KUKA KRL program: EPS_2_25694_LG02A_A_20260223033037.src

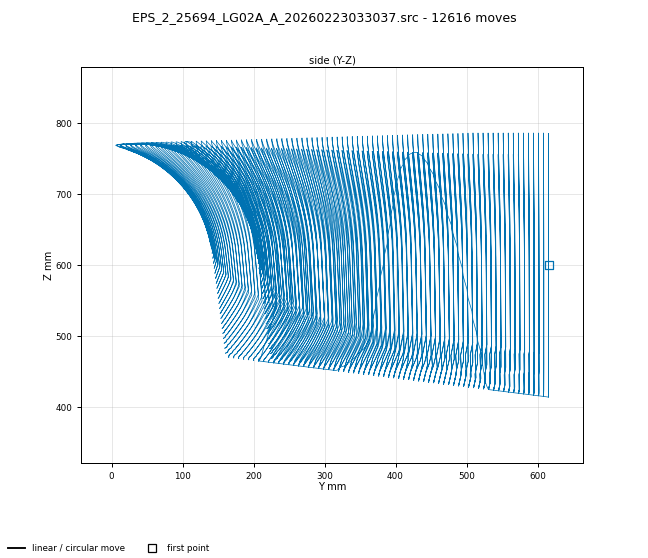
[picture p0: tool path of EPS_2_25694_LG02A_A_20260223033037.src, 12616 of 12618 moves have a stored position in this frame; points joined in program order, loops and branches not executed]
&ACCESS RVP
&REL 4
&COMMENT QRS 19112012
&PARAM EDITMASK = *
DEF PART()
EXT BAS (BAS_COMMAND :IN,REAL :IN )
INT I
BAS (#INITMOV,0 )

;KUKA QRS Post kuka4.cps  Date:22-06-2017 !

File_ID=3041

QRS_PRE_INIT()

;Init var - Until changes are made in qrs_pre_init
Outlet_Square_prg=0
Inlet_1_Square_prg=0
Inlet_2_Square_prg=0
Inlet_3_Square_prg=0
Inlet_4_Square_prg=0
Inlet_5_Square_prg=0

Outlet_1={X 0.000, Y 512.360, Z 637.000, B 0.000, E1 0.000 }
Inlet_1={X 0.000, Y 514.550, Z 607.000, B 0.000, E1 158.000 }
Outlet_1_type=299
Inlet_1_type=299
;QRS#1=Sidecore dimensions
;QRS#2=300-12" PVC SDR 35
;QRS#3=300-12" PVC SDR 35
;QRS#4=
;QRS#5=
;QRS#6=
;QRS#7=
;QRS#8=
;QRS#9=16M PSX
;QRS#10=16M PSX
;QRS#11=
;QRS#12=
;QRS#13=
;QRS#14=
;QRS#15=
;QRS#16=1220x127x1067 3,5'
;QRS#17=EPS Height
;QRS#18=786,5
;QRS#19=*
;QRS#20= UPDATED VERSION 22-06-2017
;QRS#21=*
Outlet_Square=0150
Inlet_1_Square=0150
Inlet_2_Square=0
Inlet_3_Square=0
Inlet_4_Square=0
Inlet_5_Square=0
Mill_Square=1
Outlet_Square_Prg=206
Inlet_1_Square_prg=206

QRS_INIT()

$ADVANCE=5

; T1
PTP {E1 173.596,E2 173.596}
PTP {X 0,Y 615.509,A -85,B 0,C 180,E1 173.596,E2 173.596,E3 0,E4 0,E5 0,E6 0}
QRS_SPEED_INIT()
LIN {X 0,Y 615.509,Z 600,A -85,B 0,C 180,E1 173.596,E2 173.596,E3 0,E4 0,E5 0,E6 0} C_VEL
LIN {X 0,Y 615.509,Z 424.501,A -85,B 0,C 180,E1 173.596,E2 173.596} C_VEL
LIN {X 0,Y 615.509,Z 416.32,A -85,B 0,C 180,E1 173.596,E2 173.596} C_VEL
LIN {X 0,Y 615.491,Z 414.32,A -85,B 0,C 180,E1 173.41,E2 173.41} C_VEL
LIN {X 0,Y 615.479,Z 414.31,A -85,B 0,C 180,E1 170.801,E2 170.801} C_VEL
LIN {X 0,Y 615.485,Z 414.312,A -85,B 0,C 180,E1 168.139,E2 168.139} C_VEL
LIN {X 0,Y 615.494,Z 414.321,A -85,B 0,C 180,E1 165.451,E2 165.451} C_VEL
LIN {X 0,Y 615.478,Z 414.309,A -85,B 0,C 180,E1 162.729,E2 162.729} C_VEL
LIN {X 0,Y 615.483,Z 414.316,A -85,B 0,C 180,E1 159.967,E2 159.967} C_VEL
LIN {X 0,Y 615.482,Z 414.315,A -85,B 0,C 180,E1 157.155,E2 157.155} C_VEL
LIN {X 0,Y 615.495,Z 414.307,A -85,B 0,C 180,E1 154.284,E2 154.284} C_VEL
LIN {X 0,Y 615.491,Z 414.319,A -85,B 0,C 180,E1 151.342,E2 151.342} C_VEL
LIN {X 0,Y 615.477,Z 414.312,A -85,B 0,C 180,E1 148.914,E2 148.914} C_VEL
LIN {X 0,Y 615.485,Z 414.307,A -85,B 0,C 180,E1 146.464,E2 146.464} C_VEL
LIN {X 0,Y 615.491,Z 414.326,A -85,B 0,C 180,E1 143.575,E2 143.575} C_VEL
LIN {X 0,Y 615.479,Z 414.312,A -85,B 0,C 180,E1 140.938,E2 140.938} C_VEL
LIN {X 0,Y 615.482,Z 414.308,A -85,B 0,C 180,E1 138.525,E2 138.525} C_VEL
LIN {X 0,Y 615.484,Z 414.318,A -85,B 0,C 180,E1 135.85,E2 135.85} C_VEL
LIN {X 0,Y 615.492,Z 414.493,A -85,B 0,C 180,E1 134.245,E2 134.245} C_VEL
LIN {X 0,Y 615.492,Z 437.328,A -85,B 0,C 180,E1 131.283,E2 131.283} C_VEL
LIN {X 0,Y 615.491,Z 445.894,A -85,B 0,C 180,E1 130.186,E2 130.186} C_VEL
LIN {X 0,Y 615.498,Z 610.513,A -85,B 0,C 180,E1 128.197,E2 128.197} C_VEL
LIN {X 0,Y 615.48,Z 626.456,A -85,B 0,C 180,E1 127.867,E2 127.867} C_VEL
LIN {X 0,Y 615.485,Z 642.268,A -85,B 0,C 180,E1 127.385,E2 127.385} C_VEL
LIN {X 0,Y 615.486,Z 656.531,A -85,B 0,C 180,E1 126.809,E2 126.809} C_VEL
LIN {X 0,Y 615.498,Z 671.233,A -85,B 0,C 180,E1 126.055,E2 126.055} C_VEL
LIN {X 0,Y 615.497,Z 684.53,A -85,B 0,C 180,E1 125.213,E2 125.213} C_VEL
LIN {X 0,Y 615.497,Z 695.772,A -85,B 0,C 180,E1 124.36,E2 124.36} C_VEL
LIN {X 0,Y 615.497,Z 706.636,A -85,B 0,C 180,E1 123.385,E2 123.385} C_VEL
LIN {X 0,Y 615.496,Z 716.523,A -85,B 0,C 180,E1 122.332,E2 122.332} C_VEL
LIN {X 0,Y 615.497,Z 725.201,A -85,B 0,C 180,E1 121.235,E2 121.235} C_VEL
LIN {X 0,Y 615.497,Z 733.498,A -85,B 0,C 180,E1 119.977,E2 119.977} C_VEL
LIN {X 0,Y 615.493,Z 740.563,A -85,B 0,C 180,E1 118.657,E2 118.657} C_VEL
LIN {X 0,Y 615.496,Z 745.364,A -85,B 0,C 180,E1 117.544,E2 117.544} C_VEL
LIN {X 0,Y 615.49,Z 749.169,A -85,B 0,C 180,E1 116.443,E2 116.443} C_VEL
LIN {X 0,Y 615.491,Z 751.577,A -85,B 0,C 180,E1 115.569,E2 115.569} C_VEL
LIN {X 0,Y 615.495,Z 754.487,A -85,B 0,C 180,E1 114.009,E2 114.009} C_VEL
LIN {X 0,Y 615.491,Z 755.603,A -85,B 0,C 180,E1 112.844,E2 112.844} C_VEL
LIN {X 0,Y 615.494,Z 755.77,A -85,B 0,C 180,E1 111.431,E2 111.431} C_VEL
LIN {X 0,Y 615.492,Z 754.641,A -85,B 0,C 180,E1 110.032,E2 110.032} C_VEL
LIN {X 0,Y 615.488,Z 752.15,A -85,B 0,C 180,E1 108.604,E2 108.604} C_VEL
LIN {X 0,Y 615.49,Z 748.538,A -85,B 0,C 180,E1 107.27,E2 107.27} C_VEL
LIN {X 0,Y 615.495,Z 743.488,A -85,B 0,C 180,E1 105.904,E2 105.904} C_VEL
LIN {X 0,Y 615.492,Z 736.984,A -85,B 0,C 180,E1 104.548,E2 104.548} C_VEL
LIN {X 0,Y 615.494,Z 729.996,A -85,B 0,C 180,E1 103.369,E2 103.369} C_VEL
LIN {X 0,Y 615.494,Z 721.605,A -85,B 0,C 180,E1 102.195,E2 102.195} C_VEL
LIN {X 0,Y 615.499,Z 711.689,A -85,B 0,C 180,E1 101.041,E2 101.041} C_VEL
LIN {X 0,Y 615.497,Z 701.323,A -85,B 0,C 180,E1 100.028,E2 100.028} C_VEL
LIN {X 0,Y 615.497,Z 689.159,A -85,B 0,C 180,E1 99.033,E2 99.033} C_VEL
LIN {X 0,Y 615.498,Z 677.091,A -85,B 0,C 180,E1 98.205,E2 98.205} C_VEL
LIN {X 0,Y 615.482,Z 664.005,A -85,B 0,C 180,E1 97.463,E2 97.463} C_VEL
LIN {X 0,Y 615.493,Z 648.849,A -85,B 0,C 180,E1 96.774,E2 96.774} C_VEL
LIN {X 0,Y 615.487,Z 634.492,A -85,B 0,C 180,E1 96.268,E2 96.268} C_VEL
LIN {X 0,Y 615.499,Z 620.216,A -85,B 0,C 180,E1 95.898,E2 95.898} C_VEL
LIN {X 0,Y 615.479,Z 604.737,A -85,B 0,C 180,E1 95.631,E2 95.631} C_VEL
LIN {X 0,Y 615.479,Z 445.887,A -85,B 0,C 180,E1 93.723,E2 93.723} C_VEL
LIN {X 0,Y 615.493,Z 424.588,A -85,B 0,C 180,E1 90.981,E2 90.981} C_VEL
LIN {X 0,Y 615.478,Z 414.31,A -85,B 0,C 180,E1 89.632,E2 89.632} C_VEL
LIN {X 0,Y 615.476,Z 414.309,A -85,B 0,C 180,E1 87.382,E2 87.382} C_VEL
LIN {X 0,Y 615.488,Z 414.315,A -85,B 0,C 180,E1 84.759,E2 84.759} C_VEL
LIN {X 0,Y 615.496,Z 414.317,A -85,B 0,C 180,E1 82.124,E2 82.124} C_VEL
LIN {X 0,Y 615.476,Z 414.31,A -85,B 0,C 180,E1 79.473,E2 79.473} C_VEL
LIN {X 0,Y 615.493,Z 414.312,A -85,B 0,C 180,E1 76.799,E2 76.799} C_VEL
LIN {X 0,Y 615.495,Z 414.316,A -85,B 0,C 180,E1 74.095,E2 74.095} C_VEL
LIN {X 0,Y 615.477,Z 414.309,A -85,B 0,C 180,E1 71.353,E2 71.353} C_VEL
LIN {X 0,Y 615.494,Z 414.319,A -85,B 0,C 180,E1 68.568,E2 68.568} C_VEL
LIN {X 0,Y 615.488,Z 414.31,A -85,B 0,C 180,E1 65.728,E2 65.728} C_VEL
LIN {X 0,Y 615.491,Z 414.309,A -85,B 0,C 180,E1 62.955,E2 62.955} C_VEL
LIN {X 0,Y 615.494,Z 414.321,A -85,B 0,C 180,E1 60.205,E2 60.205} C_VEL
LIN {X 0,Y 615.481,Z 414.309,A -85,B 0,C 180,E1 57.542,E2 57.542} C_VEL
LIN {X 0,Y 615.478,Z 414.309,A -85,B 0,C 180,E1 55.184,E2 55.184} C_VEL
LIN {X 0,Y 615.494,Z 414.313,A -85,B 0,C 180,E1 52.758,E2 52.758} C_VEL
LIN {X 0,Y 615.494,Z 414.312,A -85,B 0,C 180,E1 49.911,E2 49.911} C_VEL
LIN {X 0,Y 615.49,Z 414.308,A -85,B 0,C 180,E1 47.647,E2 47.647} C_VEL
LIN {X 0,Y 615.482,Z 414.312,A -85,B 0,C 180,E1 44.931,E2 44.931} C_VEL
LIN {X 0,Y 615.49,Z 414.318,A -85,B 0,C 180,E1 42.081,E2 42.081} C_VEL
LIN {X 0,Y 615.498,Z 414.308,A -85,B 0,C 180,E1 39.75,E2 39.75} C_VEL
LIN {X 0,Y 615.479,Z 414.312,A -85,B 0,C 180,E1 36.936,E2 36.936} C_VEL
LIN {X 0,Y 615.493,Z 414.314,A -85,B 0,C 180,E1 34.702,E2 34.702} C_VEL
LIN {X 0,Y 615.488,Z 414.309,A -85,B 0,C 180,E1 31.686,E2 31.686} C_VEL
LIN {X 0,Y 615.482,Z 414.308,A -85,B 0,C 180,E1 29.407,E2 29.407} C_VEL
LIN {X 0,Y 615.478,Z 414.311,A -85,B 0,C 180,E1 27.044,E2 27.044} C_VEL
LIN {X 0,Y 615.492,Z 414.325,A -85,B 0,C 180,E1 24.272,E2 24.272} C_VEL
LIN {X 0,Y 615.486,Z 414.307,A -85,B 0,C 180,E1 21.432,E2 21.432} C_VEL
LIN {X 0,Y 615.494,Z 414.316,A -85,B 0,C 180,E1 18.607,E2 18.607} C_VEL
LIN {X 0,Y 615.487,Z 414.314,A -85,B 0,C 180,E1 15.905,E2 15.905} C_VEL
LIN {X 0,Y 615.478,Z 414.309,A -85,B 0,C 180,E1 13.202,E2 13.202} C_VEL
LIN {X 0,Y 615.494,Z 414.319,A -85,B 0,C 180,E1 10.527,E2 10.527} C_VEL
LIN {X 0,Y 615.486,Z 414.314,A -85,B 0,C 180,E1 7.876,E2 7.876} C_VEL
LIN {X 0,Y 615.481,Z 414.308,A -85,B 0,C 180,E1 5.241,E2 5.241} C_VEL
LIN {X 0,Y 615.491,Z 414.316,A -85,B 0,C 180,E1 2.618,E2 2.618} C_VEL
LIN {X 0,Y 615.486,Z 414.317,A -85,B 0,C 180,E1 0,E2 0} C_VEL
LIN {X 0,Y 615.491,Z 414.306,A -85,B 0,C 180,E1 -2.618,E2 -2.618} C_VEL
LIN {X 0,Y 615.477,Z 414.316,A -85,B 0,C 180,E1 -5.241,E2 -5.241} C_VEL
LIN {X 0,Y 615.489,Z 414.321,A -85,B 0,C 180,E1 -7.875,E2 -7.875} C_VEL
LIN {X 0,Y 615.489,Z 414.307,A -85,B 0,C 180,E1 -10.527,E2 -10.527} C_VEL
LIN {X 0,Y 615.478,Z 414.314,A -85,B 0,C 180,E1 -13.201,E2 -13.201} C_VEL
LIN {X 0,Y 615.487,Z 414.32,A -85,B 0,C 180,E1 -15.905,E2 -15.905} C_VEL
LIN {X 0,Y 615.49,Z 414.306,A -85,B 0,C 180,E1 -18.646,E2 -18.646} C_VEL
LIN {X 0,Y 615.486,Z 414.318,A -85,B 0,C 180,E1 -21.432,E2 -21.432} C_VEL
LIN {X 0,Y 615.481,Z 414.312,A -85,B 0,C 180,E1 -24.272,E2 -24.272} C_VEL
LIN {X 0,Y 615.478,Z 414.311,A -85,B 0,C 180,E1 -27.044,E2 -27.044} C_VEL
LIN {X 0,Y 615.492,Z 414.324,A -85,B 0,C 180,E1 -29.796,E2 -29.796} C_VEL
LIN {X 0,Y 615.485,Z 414.309,A -85,B 0,C 180,E1 -32.458,E2 -32.458} C_VEL
LIN {X 0,Y 615.49,Z 414.306,A -85,B 0,C 180,E1 -34.815,E2 -34.815} C_VEL
LIN {X 0,Y 615.477,Z 414.315,A -85,B 0,C 180,E1 -37.243,E2 -37.243} C_VEL
LIN {X 0,Y 615.478,Z 414.317,A -85,B 0,C 180,E1 -40.088,E2 -40.088} C_VEL
LIN {X 0,Y 615.478,Z 414.312,A -85,B 0,C 180,E1 -42.354,E2 -42.354} C_VEL
LIN {X 0,Y 615.481,Z 414.311,A -85,B 0,C 180,E1 -45.069,E2 -45.069} C_VEL
LIN {X 0,Y 615.488,Z 414.32,A -85,B 0,C 180,E1 -47.92,E2 -47.92} C_VEL
LIN {X 0,Y 615.477,Z 414.314,A -85,B 0,C 180,E1 -50.249,E2 -50.249} C_VEL
LIN {X 0,Y 615.483,Z 414.31,A -85,B 0,C 180,E1 -53.064,E2 -53.064} C_VEL
LIN {X 0,Y 615.487,Z 414.319,A -85,B 0,C 180,E1 -55.978,E2 -55.978} C_VEL
LIN {X 0,Y 615.476,Z 414.313,A -85,B 0,C 180,E1 -58.314,E2 -58.314} C_VEL
LIN {X 0,Y 615.478,Z 414.309,A -85,B 0,C 180,E1 -60.593,E2 -60.593} C_VEL
LIN {X 0,Y 615.492,Z 414.307,A -85,B 0,C 180,E1 -62.954,E2 -62.954} C_VEL
LIN {X 0,Y 615.493,Z 414.437,A -85,B 0,C 180,E1 -64.937,E2 -64.937} C_VEL
LIN {X 0,Y 615.495,Z 440.026,A -85,B 0,C 180,E1 -67.864,E2 -67.864} C_VEL
LIN {X 0,Y 615.49,Z 466.555,A -85,B 0,C 180,E1 -70.835,E2 -70.835} C_VEL
LIN {X 0,Y 615.487,Z 474.978,A -85,B 0,C 180,E1 -71.761,E2 -71.761} C_VEL
LIN {X 0,Y 615.485,Z 641.166,A -85,B 0,C 180,E1 -73.768,E2 -73.768} C_VEL
LIN {X 0,Y 615.487,Z 656.706,A -85,B 0,C 180,E1 -74.095,E2 -74.095} C_VEL
LIN {X 0,Y 615.479,Z 672.046,A -85,B 0,C 180,E1 -74.562,E2 -74.562} C_VEL
LIN {X 0,Y 615.484,Z 685.749,A -85,B 0,C 180,E1 -75.112,E2 -75.112} C_VEL
LIN {X 0,Y 615.493,Z 700.045,A -85,B 0,C 180,E1 -75.833,E2 -75.833} C_VEL
LIN {X 0,Y 615.497,Z 712.896,A -85,B 0,C 180,E1 -76.631,E2 -76.631} C_VEL
LIN {X 0,Y 615.495,Z 725.252,A -85,B 0,C 180,E1 -77.554,E2 -77.554} C_VEL
LIN {X 0,Y 615.495,Z 735.604,A -85,B 0,C 180,E1 -78.473,E2 -78.473} C_VEL
LIN {X 0,Y 615.494,Z 745.182,A -85,B 0,C 180,E1 -79.473,E2 -79.473} C_VEL
LIN {X 0,Y 615.495,Z 754.575,A -85,B 0,C 180,E1 -80.635,E2 -80.635} C_VEL
LIN {X 0,Y 615.495,Z 762.379,A -85,B 0,C 180,E1 -81.794,E2 -81.794} C_VEL
LIN {X 0,Y 615.497,Z 769.606,A -85,B 0,C 180,E1 -83.102,E2 -83.102} C_VEL
LIN {X 0,Y 615.499,Z 775.435,A -85,B 0,C 180,E1 -84.43,E2 -84.43} C_VEL
LIN {X 0,Y 615.491,Z 778.859,A -85,B 0,C 180,E1 -85.415,E2 -85.415} C_VEL
LIN {X 0,Y 615.492,Z 782.317,A -85,B 0,C 180,E1 -86.727,E2 -86.727} C_VEL
LIN {X 0,Y 615.495,Z 784.593,A -85,B 0,C 180,E1 -88.037,E2 -88.037} C_VEL
LIN {X 0,Y 615.493,Z 785.74,A -85,B 0,C 180,E1 -89.345,E2 -89.345} C_VEL
LIN {X 0,Y 615.493,Z 785.741,A -85,B 0,C 180,E1 -90.654,E2 -90.654} C_VEL
LIN {X 0,Y 615.495,Z 784.594,A -85,B 0,C 180,E1 -91.963,E2 -91.963} C_VEL
LIN {X 0,Y 615.492,Z 782.319,A -85,B 0,C 180,E1 -93.273,E2 -93.273} C_VEL
LIN {X 0,Y 615.491,Z 778.862,A -85,B 0,C 180,E1 -94.584,E2 -94.584} C_VEL
LIN {X 0,Y 615.49,Z 774.145,A -85,B 0,C 180,E1 -95.898,E2 -95.898} C_VEL
LIN {X 0,Y 615.496,Z 768.031,A -85,B 0,C 180,E1 -97.215,E2 -97.215} C_VEL
LIN {X 0,Y 615.49,Z 760.336,A -85,B 0,C 180,E1 -98.536,E2 -98.536} C_VEL
LIN {X 0,Y 615.495,Z 752.117,A -85,B 0,C 180,E1 -99.696,E2 -99.696} C_VEL
LIN {X 0,Y 615.496,Z 741.897,A -85,B 0,C 180,E1 -100.892,E2 -100.892} C_VEL
LIN {X 0,Y 615.495,Z 732.073,A -85,B 0,C 180,E1 -101.86,E2 -101.86} C_VEL
LIN {X 0,Y 615.497,Z 719.954,A -85,B 0,C 180,E1 -102.865,E2 -102.865} C_VEL
LIN {X 0,Y 615.498,Z 707.806,A -85,B 0,C 180,E1 -103.705,E2 -103.705} C_VEL
LIN {X 0,Y 615.477,Z 694.388,A -85,B 0,C 180,E1 -104.472,E2 -104.472} C_VEL
LIN {X 0,Y 615.495,Z 679.86,A -85,B 0,C 180,E1 -105.141,E2 -105.141} C_VEL
LIN {X 0,Y 615.477,Z 665.632,A -85,B 0,C 180,E1 -105.65,E2 -105.65} C_VEL
LIN {X 0,Y 615.495,Z 651.159,A -85,B 0,C 180,E1 -106.035,E2 -106.035} C_VEL
LIN {X 0,Y 615.485,Z 636.616,A -85,B 0,C 180,E1 -106.297,E2 -106.297} C_VEL
LIN {X 0,Y 615.49,Z 474.74,A -85,B 0,C 180,E1 -108.259,E2 -108.259} C_VEL
LIN {X 0,Y 615.496,Z 449.397,A -85,B 0,C 180,E1 -111.08,E2 -111.08} C_VEL
LIN {X 0,Y 615.491,Z 423.588,A -85,B 0,C 180,E1 -114.009,E2 -114.009} C_VEL
LIN {X 0,Y 615.491,Z 414.306,A -85,B 0,C 180,E1 -115.099,E2 -115.099} C_VEL
LIN {X 0,Y 615.483,Z 414.317,A -85,B 0,C 180,E1 -117.915,E2 -117.915} C_VEL
LIN {X 0,Y 615.499,Z 414.321,A -85,B 0,C 180,E1 -120.159,E2 -120.159} C_VEL
LIN {X 0,Y 615.487,Z 414.321,A -85,B 0,C 180,E1 -122.457,E2 -122.457} C_VEL
LIN {X 0,Y 615.481,Z 414.313,A -85,B 0,C 180,E1 -124.815,E2 -124.815} C_VEL
LIN {X 0,Y 615.491,Z 414.306,A -85,B 0,C 180,E1 -127.241,E2 -127.241} C_VEL
LIN {X 0,Y 615.489,Z 414.32,A -85,B 0,C 180,E1 -130.089,E2 -130.089} C_VEL
LIN {X 0,Y 615.487,Z 414.308,A -85,B 0,C 180,E1 -133.047,E2 -133.047} C_VEL
LIN {X 0,Y 615.482,Z 414.318,A -85,B 0,C 180,E1 -136.002,E2 -136.002} C_VEL
LIN {X 0,Y 615.479,Z 414.312,A -85,B 0,C 180,E1 -138.905,E2 -138.905} C_VEL
LIN {X 0,Y 615.484,Z 414.308,A -85,B 0,C 180,E1 -141.096,E2 -141.096} C_VEL
LIN {X 0,Y 615.481,Z 414.31,A -85,B 0,C 180,E1 -143.575,E2 -143.575} C_VEL
LIN {X 0,Y 615.479,Z 414.318,A -85,B 0,C 180,E1 -145.978,E2 -145.978} C_VEL
LIN {X 0,Y 615.485,Z 414.328,A -85,B 0,C 180,E1 -148.315,E2 -148.315} C_VEL
LIN {X 0,Y 615.482,Z 414.319,A -85,B 0,C 180,E1 -150.594,E2 -150.594} C_VEL
LIN {X 0,Y 615.478,Z 414.312,A -85,B 0,C 180,E1 -152.955,E2 -152.955} C_VEL
LIN {X 0,Y 615.479,Z 414.312,A -85,B 0,C 180,E1 -155.728,E2 -155.728} C_VEL
LIN {X 0,Y 615.486,Z 414.32,A -85,B 0,C 180,E1 -158.568,E2 -158.568} C_VEL
LIN {X 0,Y 615.492,Z 414.306,A -85,B 0,C 180,E1 -161.391,E2 -161.391} C_VEL
LIN {X 0,Y 615.484,Z 414.319,A -85,B 0,C 180,E1 -164.095,E2 -164.095} C_VEL
LIN {X 0,Y 615.478,Z 414.315,A -85,B 0,C 180,E1 -166.799,E2 -166.799} C_VEL
LIN {X 0,Y 615.489,Z 414.307,A -85,B 0,C 180,E1 -169.473,E2 -169.473} C_VEL
LIN {X 0,Y 615.485,Z 414.32,A -85,B 0,C 180,E1 -172.124,E2 -172.124} C_VEL
LIN {X 0,Y 615.477,Z 414.317,A -85,B 0,C 180,E1 -174.759,E2 -174.759} C_VEL
LIN {X 0,Y 615.491,Z 414.306,A -85,B 0,C 180,E1 -177.382,E2 -177.382} C_VEL
LIN {X 0,Y 615.479,Z 414.317,A -85,B 0,C 180,E1 -180,E2 -180} C_VEL
LIN {X 0,Y 615.491,Z 414.318,A -85,B 0,C 180,E1 -182.618,E2 -182.618} C_VEL
LIN {X 0,Y 615.477,Z 414.31,A -85,B 0,C 180,E1 -185.241,E2 -185.241} C_VEL
LIN {X 0,Y 615.491,Z 414.32,A -85,B 0,C 180,E1 -186.59,E2 -186.59} C_VEL
LIN {X 0,Y 614.807,Z 414.458,A -85,B 0,C 180,E1 -187.136,E2 -187.136} C_VEL
LIN {X 0,Y 611.965,Z 414.879,A -85,B 0,C 180,E1 -188.022,E2 -188.022} C_VEL
LIN {X 0,Y 609.573,Z 415.186,A -85,B 0,C 180,E1 -188.734,E2 -188.734} C_VEL
LIN {X 0,Y 608.541,Z 415.302,A -85,B 0,C 180,E1 -189.284,E2 -189.284} C_VEL
LIN {X 0,Y 608.453,Z 415.312,A -85,B 0,C 180,E1 -189.47,E2 -189.47} C_VEL
LIN {X 0,Y 608.462,Z 415.315,A -85,B 0,C 180,E1 -192,E2 -192} C_VEL
LIN {X 0,Y 608.477,Z 415.314,A -85,B 0,C 180,E1 -194.721,E2 -194.721} C_VEL
LIN {X 0,Y 608.447,Z 415.313,A -85,B 0,C 180,E1 -197.477,E2 -197.477} C_VEL
LIN {X 0,Y 608.464,Z 415.319,A -85,B 0,C 180,E1 -200.274,E2 -200.274} C_VEL
LIN {X 0,Y 608.473,Z 415.32,A -85,B 0,C 180,E1 -202.482,E2 -202.482} C_VEL
LIN {X 0,Y 608.451,Z 415.312,A -85,B 0,C 180,E1 -205.301,E2 -205.301} C_VEL
LIN {X 0,Y 608.445,Z 415.313,A -85,B 0,C 180,E1 -207.518,E2 -207.518} C_VEL
LIN {X 0,Y 608.469,Z 415.313,A -85,B 0,C 180,E1 -209.974,E2 -209.974} C_VEL
LIN {X 0,Y 608.469,Z 415.32,A -85,B 0,C 180,E1 -212.525,E2 -212.525} C_VEL
LIN {X 0,Y 608.449,Z 415.313,A -85,B 0,C 180,E1 -215.278,E2 -215.278} C_VEL
LIN {X 0,Y 608.467,Z 415.318,A -85,B 0,C 180,E1 -218.242,E2 -218.242} C_VEL
LIN {X 0,Y 608.478,Z 415.318,A -85,B 0,C 180,E1 -220.333,E2 -220.333} C_VEL
LIN {X 0,Y 608.464,Z 415.311,A -85,B 0,C 180,E1 -223.309,E2 -223.309} C_VEL
LIN {X 0,Y 608.475,Z 415.41,A -85,B 0,C 180,E1 -225.605,E2 -225.605} C_VEL
LIN {X 0,Y 608.559,Z 433.198,A -85,B 0,C 180,E1 -227.948,E2 -227.948} C_VEL
LIN {X 0,Y 608.526,Z 445.944,A -85,B 0,C 180,E1 -229.602,E2 -229.602} C_VEL
LIN {X 0,Y 608.759,Z 460.794,A -85,B 0,C 180,E1 -229.79,E2 -229.79} C_VEL
LIN {X 0,Y 608.685,Z 611.468,A -85,B 0,C 180,E1 -231.632,E2 -231.632} C_VEL
LIN {X 0,Y 608.638,Z 626.926,A -85,B 0,C 180,E1 -231.962,E2 -231.962} C_VEL
LIN {X 0,Y 608.619,Z 642.036,A -85,B 0,C 180,E1 -232.428,E2 -232.428} C_VEL
LIN {X 0,Y 608.597,Z 656.166,A -85,B 0,C 180,E1 -233.003,E2 -233.003} C_VEL
LIN {X 0,Y 608.573,Z 670.032,A -85,B 0,C 180,E1 -233.712,E2 -233.712} C_VEL
LIN {X 0,Y 608.537,Z 683.04,A -85,B 0,C 180,E1 -234.527,E2 -234.527} C_VEL
LIN {X 0,Y 608.511,Z 694.952,A -85,B 0,C 180,E1 -235.422,E2 -235.422} C_VEL
LIN {X 0,Y 608.503,Z 706.251,A -85,B 0,C 180,E1 -236.432,E2 -236.432} C_VEL
LIN {X 0,Y 608.471,Z 716.109,A -85,B 0,C 180,E1 -237.477,E2 -237.477} C_VEL
LIN {X 0,Y 608.455,Z 726.038,A -85,B 0,C 180,E1 -238.732,E2 -238.732} C_VEL
LIN {X 0,Y 608.463,Z 734.461,A -85,B 0,C 180,E1 -240.03,E2 -240.03} C_VEL
LIN {X 0,Y 608.43,Z 741.587,A -85,B 0,C 180,E1 -241.388,E2 -241.388} C_VEL
LIN {X 0,Y 608.432,Z 747.381,A -85,B 0,C 180,E1 -242.802,E2 -242.802} C_VEL
LIN {X 0,Y 608.429,Z 751.003,A -85,B 0,C 180,E1 -243.964,E2 -243.964} C_VEL
LIN {X 0,Y 608.416,Z 754.237,A -85,B 0,C 180,E1 -245.428,E2 -245.428} C_VEL
LIN {X 0,Y 608.429,Z 756.021,A -85,B 0,C 180,E1 -246.876,E2 -246.876} C_VEL
LIN {X 0,Y 608.415,Z 756.445,A -85,B 0,C 180,E1 -248.307,E2 -248.307} C_VEL
LIN {X 0,Y 608.431,Z 755.551,A -85,B 0,C 180,E1 -249.725,E2 -249.725} C_VEL
LIN {X 0,Y 608.424,Z 753.375,A -85,B 0,C 180,E1 -251.13,E2 -251.13} C_VEL
LIN {X 0,Y 608.425,Z 749.892,A -85,B 0,C 180,E1 -252.523,E2 -252.523} C_VEL
LIN {X 0,Y 608.459,Z 745.057,A -85,B 0,C 180,E1 -253.907,E2 -253.907} C_VEL
LIN {X 0,Y 608.453,Z 738.775,A -85,B 0,C 180,E1 -255.28,E2 -255.28} C_VEL
LIN {X 0,Y 608.46,Z 730.901,A -85,B 0,C 180,E1 -256.644,E2 -256.644} C_VEL
LIN {X 0,Y 608.482,Z 722.538,A -85,B 0,C 180,E1 -257.832,E2 -257.832} C_VEL
LIN {X 0,Y 608.504,Z 712.409,A -85,B 0,C 180,E1 -259.029,E2 -259.029} C_VEL
LIN {X 0,Y 608.492,Z 702.409,A -85,B 0,C 180,E1 -260.024,E2 -260.024} C_VEL
LIN {X 0,Y 608.518,Z 690.408,A -85,B 0,C 180,E1 -261.031,E2 -261.031} C_VEL
LIN {X 0,Y 608.557,Z 677.176,A -85,B 0,C 180,E1 -261.951,E2 -261.951} C_VEL
LIN {X 0,Y 608.585,Z 664.061,A -85,B 0,C 180,E1 -262.703,E2 -262.703} C_VEL
LIN {X 0,Y 608.61,Z 649.663,A -85,B 0,C 180,E1 -263.369,E2 -263.369} C_VEL
LIN {X 0,Y 608.642,Z 634.561,A -85,B 0,C 180,E1 -263.911,E2 -263.911} C_VEL
LIN {X 0,Y 608.695,Z 619.386,A -85,B 0,C 180,E1 -264.306,E2 -264.306} C_VEL
LIN {X 0,Y 608.688,Z 603.326,A -85,B 0,C 180,E1 -264.576,E2 -264.576} C_VEL
LIN {X 0,Y 608.664,Z 446.816,A -85,B 0,C 180,E1 -266.473,E2 -266.473} C_VEL
LIN {X 0,Y 608.518,Z 445.667,A -85,B 0,C 180,E1 -266.524,E2 -266.524} C_VEL
LIN {X 0,Y 608.58,Z 425.315,A -85,B 0,C 180,E1 -269.173,E2 -269.173} C_VEL
LIN {X 0,Y 608.45,Z 415.314,A -85,B 0,C 180,E1 -270.517,E2 -270.517} C_VEL
LIN {X 0,Y 608.485,Z 415.314,A -85,B 0,C 180,E1 -273.311,E2 -273.311} C_VEL
LIN {X 0,Y 608.467,Z 415.315,A -85,B 0,C 180,E1 -275.967,E2 -275.967} C_VEL
LIN {X 0,Y 608.449,Z 415.313,A -85,B 0,C 180,E1 -278.636,E2 -278.636} C_VEL
LIN {X 0,Y 608.484,Z 415.313,A -85,B 0,C 180,E1 -281.324,E2 -281.324} C_VEL
LIN {X 0,Y 608.474,Z 415.314,A -85,B 0,C 180,E1 -284.038,E2 -284.038} C_VEL
LIN {X 0,Y 608.444,Z 415.313,A -85,B 0,C 180,E1 -286.784,E2 -286.784} C_VEL
LIN {X 0,Y 608.46,Z 415.321,A -85,B 0,C 180,E1 -289.57,E2 -289.57} C_VEL
LIN {X 0,Y 608.463,Z 415.311,A -85,B 0,C 180,E1 -292.476,E2 -292.476} C_VEL
LIN {X 0,Y 608.456,Z 415.312,A -85,B 0,C 180,E1 -294.571,E2 -294.571} C_VEL
LIN {X 0,Y 608.483,Z 415.312,A -85,B 0,C 180,E1 -297.208,E2 -297.208} C_VEL
LIN {X 0,Y 608.476,Z 415.314,A -85,B 0,C 180,E1 -299.972,E2 -299.972} C_VEL
LIN {X 0,Y 608.458,Z 415.311,A -85,B 0,C 180,E1 -302.521,E2 -302.521} C_VEL
LIN {X 0,Y 608.445,Z 415.314,A -85,B 0,C 180,E1 -304.904,E2 -304.904} C_VEL
LIN {X 0,Y 608.48,Z 415.311,A -85,B 0,C 180,E1 -307.159,E2 -307.159} C_VEL
LIN {X 0,Y 608.478,Z 415.316,A -85,B 0,C 180,E1 -309.439,E2 -309.439} C_VEL
LIN {X 0,Y 608.462,Z 415.312,A -85,B 0,C 180,E1 -312.334,E2 -312.334} C_VEL
LIN {X 0,Y 608.451,Z 415.312,A -85,B 0,C 180,E1 -314.796,E2 -314.796} C_VEL
LIN {X 0,Y 608.449,Z 415.314,A -85,B 0,C 180,E1 -317.039,E2 -317.039} C_VEL
LIN {X 0,Y 608.458,Z 415.322,A -85,B 0,C 180,E1 -319.697,E2 -319.697} C_VEL
LIN {X 0,Y 608.469,Z 415.312,A -85,B 0,C 180,E1 -322.253,E2 -322.253} C_VEL
LIN {X 0,Y 608.481,Z 415.31,A -85,B 0,C 180,E1 -325.09,E2 -325.09} C_VEL
LIN {X 0,Y 608.473,Z 415.316,A -85,B 0,C 180,E1 -327.906,E2 -327.906} C_VEL
LIN {X 0,Y 608.477,Z 415.311,A -85,B 0,C 180,E1 -330.221,E2 -330.221} C_VEL
LIN {X 0,Y 608.472,Z 415.31,A -85,B 0,C 180,E1 -332.793,E2 -332.793} C_VEL
LIN {X 0,Y 608.453,Z 415.318,A -85,B 0,C 180,E1 -335.429,E2 -335.429} C_VEL
LIN {X 0,Y 608.469,Z 415.311,A -85,B 0,C 180,E1 -338.308,E2 -338.308} C_VEL
LIN {X 0,Y 608.457,Z 415.314,A -85,B 0,C 180,E1 -341.13,E2 -341.13} C_VEL
LIN {X 0,Y 608.465,Z 415.317,A -85,B 0,C 180,E1 -343.906,E2 -343.906} C_VEL
LIN {X 0,Y 608.458,Z 415.311,A -85,B 0,C 180,E1 -346.643,E2 -346.643} C_VEL
LIN {X 0,Y 608.467,Z 415.315,A -85,B 0,C 180,E1 -349.35,E2 -349.35} C_VEL
LIN {X 0,Y 608.479,Z 415.314,A -85,B 0,C 180,E1 -352.033,E2 -352.033} C_VEL
LIN {X 0,Y 608.461,Z 415.311,A -85,B 0,C 180,E1 -354.698,E2 -354.698} C_VEL
LIN {X 0,Y 608.482,Z 415.313,A -85,B 0,C 180,E1 -357.352,E2 -357.352} C_VEL
LIN {X 0,Y 608.476,Z 415.315,A -85,B 0,C 180,E1 -360,E2 -360} C_VEL
LIN {X 0,Y 608.482,Z 415.308,A -85,B 0,C 180,E1 -362.648,E2 -362.648} C_VEL
LIN {X 0,Y 608.458,Z 415.315,A -85,B 0,C 180,E1 -365.302,E2 -365.302} C_VEL
LIN {X 0,Y 608.48,Z 415.315,A -85,B 0,C 180,E1 -367.967,E2 -367.967} C_VEL
LIN {X 0,Y 608.465,Z 415.311,A -85,B 0,C 180,E1 -370.955,E2 -370.955} C_VEL
LIN {X 0,Y 608.459,Z 415.316,A -85,B 0,C 180,E1 -373.356,E2 -373.356} C_VEL
LIN {X 0,Y 608.461,Z 415.315,A -85,B 0,C 180,E1 -376.094,E2 -376.094} C_VEL
LIN {X 0,Y 608.456,Z 415.312,A -85,B 0,C 180,E1 -378.869,E2 -378.869} C_VEL
LIN {X 0,Y 608.466,Z 415.321,A -85,B 0,C 180,E1 -381.691,E2 -381.691} C_VEL
LIN {X 0,Y 608.448,Z 415.313,A -85,B 0,C 180,E1 -384.571,E2 -384.571} C_VEL
LIN {X 0,Y 608.472,Z 415.312,A -85,B 0,C 180,E1 -387.206,E2 -387.206} C_VEL
LIN {X 0,Y 608.468,Z 415.316,A -85,B 0,C 180,E1 -389.972,E2 -389.972} C_VEL
LIN {X 0,Y 608.452,Z 415.312,A -85,B 0,C 180,E1 -392.88,E2 -392.88} C_VEL
LIN {X 0,Y 608.449,Z 415.316,A -85,B 0,C 180,E1 -395.277,E2 -395.277} C_VEL
LIN {X 0,Y 608.464,Z 415.321,A -85,B 0,C 180,E1 -397.747,E2 -397.747} C_VEL
LIN {X 0,Y 608.446,Z 415.315,A -85,B 0,C 180,E1 -400.329,E2 -400.329} C_VEL
LIN {X 0,Y 608.447,Z 415.313,A -85,B 0,C 180,E1 -402.96,E2 -402.96} C_VEL
LIN {X 0,Y 608.46,Z 415.322,A -85,B 0,C 180,E1 -405.736,E2 -405.736} C_VEL
LIN {X 0,Y 608.46,Z 415.311,A -85,B 0,C 180,E1 -408.658,E2 -408.658} C_VEL
LIN {X 0,Y 608.468,Z 415.316,A -85,B 0,C 180,E1 -411.412,E2 -411.412} C_VEL
LIN {X 0,Y 608.445,Z 415.32,A -85,B 0,C 180,E1 -413.955,E2 -413.955} C_VEL
LIN {X 0,Y 608.448,Z 415.315,A -85,B 0,C 180,E1 -416.328,E2 -416.328} C_VEL
LIN {X 0,Y 608.462,Z 415.311,A -85,B 0,C 180,E1 -418.73,E2 -418.73} C_VEL
LIN {X 0,Y 608.47,Z 415.315,A -85,B 0,C 180,E1 -421.381,E2 -421.381} C_VEL
LIN {X 0,Y 608.442,Z 415.322,A -85,B 0,C 180,E1 -423.964,E2 -423.964} C_VEL
LIN {X 0,Y 608.485,Z 415.446,A -85,B 0,C 180,E1 -424.746,E2 -424.746} C_VEL
LIN {X 0,Y 608.662,Z 424.488,A -85,B 0,C 180,E1 -425.809,E2 -425.809} C_VEL
LIN {X 0,Y 608.608,Z 447.83,A -85,B 0,C 180,E1 -428.491,E2 -428.491} C_VEL
LIN {X 0,Y 608.561,Z 471.239,A -85,B 0,C 180,E1 -431.134,E2 -431.134} C_VEL
LIN {X 0,Y 608.577,Z 474.978,A -85,B 0,C 180,E1 -431.547,E2 -431.547} C_VEL
LIN {X 0,Y 608.701,Z 587.844,A -85,B 0,C 180,E1 -432.92,E2 -432.92} C_VEL
LIN {X 0,Y 608.68,Z 641.166,A -85,B 0,C 180,E1 -433.581,E2 -433.581} C_VEL
LIN {X 0,Y 608.647,Z 656.705,A -85,B 0,C 180,E1 -433.911,E2 -433.911} C_VEL
LIN {X 0,Y 608.616,Z 672.044,A -85,B 0,C 180,E1 -434.383,E2 -434.383} C_VEL
LIN {X 0,Y 608.605,Z 685.752,A -85,B 0,C 180,E1 -434.94,E2 -434.94} C_VEL
LIN {X 0,Y 608.572,Z 699.233,A -85,B 0,C 180,E1 -435.624,E2 -435.624} C_VEL
LIN {X 0,Y 608.554,Z 711.661,A -85,B 0,C 180,E1 -436.39,E2 -436.39} C_VEL
LIN {X 0,Y 608.528,Z 724.28,A -85,B 0,C 180,E1 -437.324,E2 -437.324} C_VEL
LIN {X 0,Y 608.496,Z 735.745,A -85,B 0,C 180,E1 -438.339,E2 -438.339} C_VEL
LIN {X 0,Y 608.475,Z 745.386,A -85,B 0,C 180,E1 -439.35,E2 -439.35} C_VEL
LIN {X 0,Y 608.477,Z 754.852,A -85,B 0,C 180,E1 -440.526,E2 -440.526} C_VEL
LIN {X 0,Y 608.456,Z 762.728,A -85,B 0,C 180,E1 -441.698,E2 -441.698} C_VEL
LIN {X 0,Y 608.442,Z 770.086,A -85,B 0,C 180,E1 -443.034,E2 -443.034} C_VEL
LIN {X 0,Y 608.449,Z 775.922,A -85,B 0,C 180,E1 -444.365,E2 -444.365} C_VEL
LIN {X 0,Y 608.427,Z 779.382,A -85,B 0,C 180,E1 -445.362,E2 -445.362} C_VEL
LIN {X 0,Y 608.421,Z 782.885,A -85,B 0,C 180,E1 -446.689,E2 -446.689} C_VEL
LIN {X 0,Y 608.44,Z 785.191,A -85,B 0,C 180,E1 -448.014,E2 -448.014} C_VEL
LIN {X 0,Y 608.436,Z 786.35,A -85,B 0,C 180,E1 -449.338,E2 -449.338} C_VEL
LIN {X 0,Y 608.436,Z 786.351,A -85,B 0,C 180,E1 -450.661,E2 -450.661} C_VEL
LIN {X 0,Y 608.44,Z 785.192,A -85,B 0,C 180,E1 -451.985,E2 -451.985} C_VEL
LIN {X 0,Y 608.421,Z 782.886,A -85,B 0,C 180,E1 -453.311,E2 -453.311} C_VEL
LIN {X 0,Y 608.427,Z 779.384,A -85,B 0,C 180,E1 -454.637,E2 -454.637} C_VEL
LIN {X 0,Y 608.431,Z 774.609,A -85,B 0,C 180,E1 -455.967,E2 -455.967} C_VEL
LIN {X 0,Y 608.458,Z 768.428,A -85,B 0,C 180,E1 -457.299,E2 -457.299} C_VEL
LIN {X 0,Y 608.465,Z 760.657,A -85,B 0,C 180,E1 -458.635,E2 -458.635} C_VEL
LIN {X 0,Y 608.471,Z 752.374,A -85,B 0,C 180,E1 -459.809,E2 -459.809} C_VEL
LIN {X 0,Y 608.492,Z 741.654,A -85,B 0,C 180,E1 -461.063,E2 -461.063} C_VEL
LIN {X 0,Y 608.522,Z 730.28,A -85,B 0,C 180,E1 -462.167,E2 -462.167} C_VEL
LIN {X 0,Y 608.547,Z 718.861,A -85,B 0,C 180,E1 -463.099,E2 -463.099} C_VEL
LIN {X 0,Y 608.561,Z 706.455,A -85,B 0,C 180,E1 -463.95,E2 -463.95} C_VEL
LIN {X 0,Y 608.56,Z 692.87,A -85,B 0,C 180,E1 -464.718,E2 -464.718} C_VEL
LIN {X 0,Y 608.63,Z 678.805,A -85,B 0,C 180,E1 -465.358,E2 -465.358} C_VEL
LIN {X 0,Y 608.631,Z 664.319,A -85,B 0,C 180,E1 -465.874,E2 -465.874} C_VEL
LIN {X 0,Y 608.686,Z 649.039,A -85,B 0,C 180,E1 -466.269,E2 -466.269} C_VEL
LIN {X 0,Y 608.685,Z 633.11,A -85,B 0,C 180,E1 -466.534,E2 -466.534} C_VEL
LIN {X 0,Y 608.686,Z 475.642,A -85,B 0,C 180,E1 -468.442,E2 -468.442} C_VEL
LIN {X 0,Y 608.545,Z 474.565,A -85,B 0,C 180,E1 -468.495,E2 -468.495} C_VEL
LIN {X 0,Y 608.615,Z 449.397,A -85,B 0,C 180,E1 -471.33,E2 -471.33} C_VEL
LIN {X 0,Y 608.684,Z 424.44,A -85,B 0,C 180,E1 -474.196,E2 -474.196} C_VEL
LIN {X 0,Y 608.484,Z 415.453,A -85,B 0,C 180,E1 -475.253,E2 -475.253} C_VEL
LIN {X 0,Y 608.449,Z 415.314,A -85,B 0,C 180,E1 -477.517,E2 -477.517} C_VEL
LIN {X 0,Y 608.466,Z 415.316,A -85,B 0,C 180,E1 -479.971,E2 -479.971} C_VEL
LIN {X 0,Y 608.462,Z 415.318,A -85,B 0,C 180,E1 -482.522,E2 -482.522} C_VEL
LIN {X 0,Y 608.435,Z 415.314,A -85,B 0,C 180,E1 -485.277,E2 -485.277} C_VEL
LIN {X 0,Y 608.47,Z 415.312,A -85,B 0,C 180,E1 -487.745,E2 -487.745} C_VEL
LIN {X 0,Y 608.452,Z 415.323,A -85,B 0,C 180,E1 -490.329,E2 -490.329} C_VEL
LIN {X 0,Y 608.484,Z 415.308,A -85,B 0,C 180,E1 -493.31,E2 -493.31} C_VEL
LIN {X 0,Y 608.466,Z 415.318,A -85,B 0,C 180,E1 -496.13,E2 -496.13} C_VEL
LIN {X 0,Y 608.449,Z 415.315,A -85,B 0,C 180,E1 -498.823,E2 -498.823} C_VEL
LIN {X 0,Y 608.465,Z 415.311,A -85,B 0,C 180,E1 -501.412,E2 -501.412} C_VEL
LIN {X 0,Y 608.472,Z 415.314,A -85,B 0,C 180,E1 -503.95,E2 -503.95} C_VEL
LIN {X 0,Y 608.461,Z 415.322,A -85,B 0,C 180,E1 -506.329,E2 -506.329} C_VEL
LIN {X 0,Y 608.47,Z 415.314,A -85,B 0,C 180,E1 -508.727,E2 -508.727} C_VEL
LIN {X 0,Y 608.471,Z 415.31,A -85,B 0,C 180,E1 -511.378,E2 -511.378} C_VEL
LIN {X 0,Y 608.477,Z 415.319,A -85,B 0,C 180,E1 -514.276,E2 -514.276} C_VEL
LIN {X 0,Y 608.447,Z 415.315,A -85,B 0,C 180,E1 -516.876,E2 -516.876} C_VEL
LIN {X 0,Y 608.459,Z 415.313,A -85,B 0,C 180,E1 -519.726,E2 -519.726} C_VEL
LIN {X 0,Y 608.445,Z 415.321,A -85,B 0,C 180,E1 -522.523,E2 -522.523} C_VEL
LIN {X 0,Y 608.473,Z 415.309,A -85,B 0,C 180,E1 -525.28,E2 -525.28} C_VEL
LIN {X 0,Y 608.46,Z 415.316,A -85,B 0,C 180,E1 -528,E2 -528} C_VEL
LIN {X 0,Y 608.463,Z 415.316,A -85,B 0,C 180,E1 -530.694,E2 -530.694} C_VEL
LIN {X 0,Y 608.469,Z 415.31,A -85,B 0,C 180,E1 -533.368,E2 -533.368} C_VEL
LIN {X 0,Y 608.453,Z 415.317,A -85,B 0,C 180,E1 -536.026,E2 -536.026} C_VEL
LIN {X 0,Y 608.468,Z 415.316,A -85,B 0,C 180,E1 -538.676,E2 -538.676} C_VEL
LIN {X 0,Y 608.468,Z 415.31,A -85,B 0,C 180,E1 -541.324,E2 -541.324} C_VEL
LIN {X 0,Y 608.453,Z 415.316,A -85,B 0,C 180,E1 -543.974,E2 -543.974} C_VEL
LIN {X 0,Y 608.469,Z 415.316,A -85,B 0,C 180,E1 -546.633,E2 -546.633} C_VEL
LIN {X 0,Y 608.453,Z 415.312,A -85,B 0,C 180,E1 -549.47,E2 -549.47} C_VEL
LIN {X 0,Y 607.776,Z 415.402,A -85,B 0,C 180,E1 -550.023,E2 -550.023} C_VEL
LIN {X 0,Y 604.924,Z 415.757,A -85,B 0,C 180,E1 -550.92,E2 -550.92} C_VEL
LIN {X 0,Y 602.522,Z 416.057,A -85,B 0,C 180,E1 -551.641,E2 -551.641} C_VEL
LIN {X 0,Y 601.492,Z 416.186,A -85,B 0,C 180,E1 -552.198,E2 -552.198} C_VEL
LIN {X 0,Y 601.409,Z 416.193,A -85,B 0,C 180,E1 -552.386,E2 -552.386} C_VEL
LIN {X 0,Y 601.429,Z 416.19,A -85,B 0,C 180,E1 -554.897,E2 -554.897} C_VEL
LIN {X 0,Y 601.429,Z 416.189,A -85,B 0,C 180,E1 -556.986,E2 -556.986} C_VEL
LIN {X 0,Y 601.404,Z 416.192,A -85,B 0,C 180,E1 -559.81,E2 -559.81} C_VEL
LIN {X 0,Y 601.418,Z 416.196,A -85,B 0,C 180,E1 -562.608,E2 -562.608} C_VEL
LIN {X 0,Y 601.401,Z 416.194,A -85,B 0,C 180,E1 -564.879,E2 -564.879} C_VEL
LIN {X 0,Y 601.422,Z 416.19,A -85,B 0,C 180,E1 -567.868,E2 -567.868} C_VEL
LIN {X 0,Y 601.443,Z 416.191,A -85,B 0,C 180,E1 -570.163,E2 -570.163} C_VEL
LIN {X 0,Y 601.425,Z 416.194,A -85,B 0,C 180,E1 -572.718,E2 -572.718} C_VEL
LIN {X 0,Y 601.415,Z 416.19,A -85,B 0,C 180,E1 -575.116,E2 -575.116} C_VEL
LIN {X 0,Y 601.43,Z 416.187,A -85,B 0,C 180,E1 -577.42,E2 -577.42} C_VEL
LIN {X 0,Y 601.412,Z 416.193,A -85,B 0,C 180,E1 -579.995,E2 -579.995} C_VEL
LIN {X 0,Y 601.409,Z 416.197,A -85,B 0,C 180,E1 -582.671,E2 -582.671} C_VEL
LIN {X 0,Y 601.45,Z 416.274,A -85,B 0,C 180,E1 -585.445,E2 -585.445} C_VEL
LIN {X 0,Y 601.692,Z 420.354,A -85,B 0,C 180,E1 -586.001,E2 -586.001} C_VEL
LIN {X 0,Y 601.627,Z 442.433,A -85,B 0,C 180,E1 -588.923,E2 -588.923} C_VEL
LIN {X 0,Y 601.594,Z 446.098,A -85,B 0,C 180,E1 -589.383,E2 -589.383} C_VEL
LIN {X 0,Y 602.04,Z 450.336,A -85,B 0,C 180,E1 -589.45,E2 -589.45} C_VEL
LIN {X 0,Y 601.875,Z 611.182,A -85,B 0,C 180,E1 -591.436,E2 -591.436} C_VEL
LIN {X 0,Y 601.819,Z 626.993,A -85,B 0,C 180,E1 -591.776,E2 -591.776} C_VEL
LIN {X 0,Y 601.769,Z 641.813,A -85,B 0,C 180,E1 -592.237,E2 -592.237} C_VEL
LIN {X 0,Y 601.712,Z 656.988,A -85,B 0,C 180,E1 -592.865,E2 -592.865} C_VEL
LIN {X 0,Y 601.658,Z 671.217,A -85,B 0,C 180,E1 -593.612,E2 -593.612} C_VEL
LIN {X 0,Y 601.586,Z 683.971,A -85,B 0,C 180,E1 -594.431,E2 -594.431} C_VEL
LIN {X 0,Y 601.518,Z 696.282,A -85,B 0,C 180,E1 -595.381,E2 -595.381} C_VEL
LIN {X 0,Y 601.487,Z 707.241,A -85,B 0,C 180,E1 -596.39,E2 -596.39} C_VEL
LIN {X 0,Y 601.44,Z 717.279,A -85,B 0,C 180,E1 -597.486,E2 -597.486} C_VEL
LIN {X 0,Y 601.397,Z 725.513,A -85,B 0,C 180,E1 -598.549,E2 -598.549} C_VEL
LIN {X 0,Y 601.385,Z 734.01,A -85,B 0,C 180,E1 -599.859,E2 -599.859} C_VEL
LIN {X 0,Y 601.347,Z 741.195,A -85,B 0,C 180,E1 -601.227,E2 -601.227} C_VEL
LIN {X 0,Y 601.351,Z 745.123,A -85,B 0,C 180,E1 -602.13,E2 -602.13} C_VEL
LIN {X 0,Y 601.349,Z 750.257,A -85,B 0,C 180,E1 -603.634,E2 -603.634} C_VEL
LIN {X 0,Y 601.328,Z 753.776,A -85,B 0,C 180,E1 -605.119,E2 -605.119} C_VEL
LIN {X 0,Y 601.323,Z 755.824,A -85,B 0,C 180,E1 -606.586,E2 -606.586} C_VEL
LIN {X 0,Y 601.336,Z 756.5,A -85,B 0,C 180,E1 -608.039,E2 -608.039} C_VEL
LIN {X 0,Y 601.347,Z 755.847,A -85,B 0,C 180,E1 -609.476,E2 -609.476} C_VEL
LIN {X 0,Y 601.311,Z 753.9,A -85,B 0,C 180,E1 -610.898,E2 -610.898} C_VEL
LIN {X 0,Y 601.316,Z 750.645,A -85,B 0,C 180,E1 -612.31,E2 -612.31} C_VEL
LIN {X 0,Y 601.362,Z 746.051,A -85,B 0,C 180,E1 -613.712,E2 -613.712} C_VEL
LIN {X 0,Y 601.373,Z 740.046,A -85,B 0,C 180,E1 -615.102,E2 -615.102} C_VEL
LIN {X 0,Y 601.381,Z 734.167,A -85,B 0,C 180,E1 -616.205,E2 -616.205} C_VEL
LIN {X 0,Y 601.417,Z 725.695,A -85,B 0,C 180,E1 -617.515,E2 -617.515} C_VEL
LIN {X 0,Y 601.448,Z 716.422,A -85,B 0,C 180,E1 -618.702,E2 -618.702} C_VEL
LIN {X 0,Y 601.483,Z 706.867,A -85,B 0,C 180,E1 -619.736,E2 -619.736} C_VEL
LIN {X 0,Y 601.543,Z 695.697,A -85,B 0,C 180,E1 -620.756,E2 -620.756} C_VEL
LIN {X 0,Y 601.6,Z 683.545,A -85,B 0,C 180,E1 -621.688,E2 -621.688} C_VEL
LIN {X 0,Y 601.654,Z 670.258,A -85,B 0,C 180,E1 -622.534,E2 -622.534} C_VEL
LIN {X 0,Y 601.716,Z 656.795,A -85,B 0,C 180,E1 -623.234,E2 -623.234} C_VEL
LIN {X 0,Y 601.755,Z 642.767,A -85,B 0,C 180,E1 -623.817,E2 -623.817} C_VEL
LIN {X 0,Y 601.833,Z 627.322,A -85,B 0,C 180,E1 -624.304,E2 -624.304} C_VEL
LIN {X 0,Y 601.876,Z 611.93,A -85,B 0,C 180,E1 -624.64,E2 -624.64} C_VEL
LIN {X 0,Y 601.912,Z 558.752,A -85,B 0,C 180,E1 -625.312,E2 -625.312} C_VEL
LIN {X 0,Y 601.938,Z 447.796,A -85,B 0,C 180,E1 -626.675,E2 -626.675} C_VEL
LIN {X 0,Y 601.579,Z 445.741,A -85,B 0,C 180,E1 -626.735,E2 -626.735} C_VEL
LIN {X 0,Y 601.671,Z 424.784,A -85,B 0,C 180,E1 -629.498,E2 -629.498} C_VEL
LIN {X 0,Y 601.492,Z 416.701,A -85,B 0,C 180,E1 -630.586,E2 -630.586} C_VEL
LIN {X 0,Y 601.445,Z 416.189,A -85,B 0,C 180,E1 -630.67,E2 -630.67} C_VEL
LIN {X 0,Y 601.436,Z 416.193,A -85,B 0,C 180,E1 -633.35,E2 -633.35} C_VEL
LIN {X 0,Y 601.418,Z 416.193,A -85,B 0,C 180,E1 -636.037,E2 -636.037} C_VEL
LIN {X 0,Y 601.412,Z 416.19,A -85,B 0,C 180,E1 -638.738,E2 -638.738} C_VEL
LIN {X 0,Y 601.442,Z 416.193,A -85,B 0,C 180,E1 -641.458,E2 -641.458} C_VEL
LIN {X 0,Y 601.424,Z 416.19,A -85,B 0,C 180,E1 -644.206,E2 -644.206} C_VEL
LIN {X 0,Y 601.418,Z 416.19,A -85,B 0,C 180,E1 -646.986,E2 -646.986} C_VEL
LIN {X 0,Y 601.412,Z 416.197,A -85,B 0,C 180,E1 -649.809,E2 -649.809} C_VEL
LIN {X 0,Y 601.416,Z 416.189,A -85,B 0,C 180,E1 -652.683,E2 -652.683} C_VEL
LIN {X 0,Y 601.406,Z 416.19,A -85,B 0,C 180,E1 -654.879,E2 -654.879} C_VEL
LIN {X 0,Y 601.423,Z 416.194,A -85,B 0,C 180,E1 -657.867,E2 -657.867} C_VEL
LIN {X 0,Y 601.433,Z 416.189,A -85,B 0,C 180,E1 -660.164,E2 -660.164} C_VEL
LIN {X 0,Y 601.421,Z 416.188,A -85,B 0,C 180,E1 -662.715,E2 -662.715} C_VEL
LIN {X 0,Y 601.398,Z 416.193,A -85,B 0,C 180,E1 -665.112,E2 -665.112} C_VEL
LIN {X 0,Y 601.439,Z 416.192,A -85,B 0,C 180,E1 -667.419,E2 -667.419} C_VEL
LIN {X 0,Y 601.413,Z 416.194,A -85,B 0,C 180,E1 -669.995,E2 -669.995} C_VEL
LIN {X 0,Y 601.414,Z 416.189,A -85,B 0,C 180,E1 -672.67,E2 -672.67} C_VEL
LIN {X 0,Y 601.428,Z 416.195,A -85,B 0,C 180,E1 -675.482,E2 -675.482} C_VEL
LIN {X 0,Y 601.424,Z 416.188,A -85,B 0,C 180,E1 -678.407,E2 -678.407} C_VEL
LIN {X 0,Y 601.434,Z 416.187,A -85,B 0,C 180,E1 -680.875,E2 -680.875} C_VEL
LIN {X 0,Y 601.445,Z 416.195,A -85,B 0,C 180,E1 -683.734,E2 -683.734} C_VEL
LIN {X 0,Y 601.427,Z 416.187,A -85,B 0,C 180,E1 -686.686,E2 -686.686} C_VEL
LIN {X 0,Y 601.414,Z 416.19,A -85,B 0,C 180,E1 -689.057,E2 -689.057} C_VEL
LIN {X 0,Y 601.439,Z 416.191,A -85,B 0,C 180,E1 -691.373,E2 -691.373} C_VEL
LIN {X 0,Y 601.421,Z 416.191,A -85,B 0,C 180,E1 -694.131,E2 -694.131} C_VEL
LIN {X 0,Y 601.42,Z 416.187,A -85,B 0,C 180,E1 -696.589,E2 -696.589} C_VEL
LIN {X 0,Y 601.435,Z 416.193,A -85,B 0,C 180,E1 -699.478,E2 -699.478} C_VEL
LIN {X 0,Y 601.396,Z 416.192,A -85,B 0,C 180,E1 -702.311,E2 -702.311} C_VEL
LIN {X 0,Y 601.412,Z 416.19,A -85,B 0,C 180,E1 -704.408,E2 -704.408} C_VEL
LIN {X 0,Y 601.422,Z 416.191,A -85,B 0,C 180,E1 -707.172,E2 -707.172} C_VEL
LIN {X 0,Y 601.435,Z 416.193,A -85,B 0,C 180,E1 -709.905,E2 -709.905} C_VEL
LIN {X 0,Y 601.438,Z 416.186,A -85,B 0,C 180,E1 -712.615,E2 -712.615} C_VEL
LIN {X 0,Y 601.429,Z 416.191,A -85,B 0,C 180,E1 -715.308,E2 -715.308} C_VEL
LIN {X 0,Y 601.426,Z 416.193,A -85,B 0,C 180,E1 -717.991,E2 -717.991} C_VEL
LIN {X 0,Y 601.451,Z 416.184,A -85,B 0,C 180,E1 -720.669,E2 -720.669} C_VEL
LIN {X 0,Y 601.428,Z 416.192,A -85,B 0,C 180,E1 -723.349,E2 -723.349} C_VEL
LIN {X 0,Y 601.415,Z 416.193,A -85,B 0,C 180,E1 -726.037,E2 -726.037} C_VEL
LIN {X 0,Y 601.437,Z 416.186,A -85,B 0,C 180,E1 -728.737,E2 -728.737} C_VEL
LIN {X 0,Y 601.433,Z 416.193,A -85,B 0,C 180,E1 -731.458,E2 -731.458} C_VEL
LIN {X 0,Y 601.419,Z 416.191,A -85,B 0,C 180,E1 -734.205,E2 -734.205} C_VEL
LIN {X 0,Y 601.431,Z 416.188,A -85,B 0,C 180,E1 -736.986,E2 -736.986} C_VEL
LIN {X 0,Y 601.404,Z 416.199,A -85,B 0,C 180,E1 -739.809,E2 -739.809} C_VEL
LIN {X 0,Y 601.414,Z 416.189,A -85,B 0,C 180,E1 -742.606,E2 -742.606} C_VEL
LIN {X 0,Y 601.399,Z 416.191,A -85,B 0,C 180,E1 -744.879,E2 -744.879} C_VEL
LIN {X 0,Y 601.419,Z 416.196,A -85,B 0,C 180,E1 -747.867,E2 -747.867} C_VEL
LIN {X 0,Y 601.427,Z 416.191,A -85,B 0,C 180,E1 -750.164,E2 -750.164} C_VEL
LIN {X 0,Y 601.419,Z 416.188,A -85,B 0,C 180,E1 -752.715,E2 -752.715} C_VEL
LIN {X 0,Y 601.415,Z 416.191,A -85,B 0,C 180,E1 -755.115,E2 -755.115} C_VEL
LIN {X 0,Y 601.432,Z 416.192,A -85,B 0,C 180,E1 -757.419,E2 -757.419} C_VEL
LIN {X 0,Y 601.411,Z 416.195,A -85,B 0,C 180,E1 -759.995,E2 -759.995} C_VEL
LIN {X 0,Y 601.408,Z 416.19,A -85,B 0,C 180,E1 -762.671,E2 -762.671} C_VEL
LIN {X 0,Y 601.426,Z 416.194,A -85,B 0,C 180,E1 -765.482,E2 -765.482} C_VEL
LIN {X 0,Y 601.424,Z 416.189,A -85,B 0,C 180,E1 -768.407,E2 -768.407} C_VEL
LIN {X 0,Y 601.434,Z 416.194,A -85,B 0,C 180,E1 -771.529,E2 -771.529} C_VEL
LIN {X 0,Y 601.385,Z 416.195,A -85,B 0,C 180,E1 -774.245,E2 -774.245} C_VEL
LIN {X 0,Y 601.419,Z 416.189,A -85,B 0,C 180,E1 -776.686,E2 -776.686} C_VEL
LIN {X 0,Y 601.424,Z 416.189,A -85,B 0,C 180,E1 -779.058,E2 -779.058} C_VEL
LIN {X 0,Y 601.43,Z 416.192,A -85,B 0,C 180,E1 -781.373,E2 -781.373} C_VEL
LIN {X 0,Y 601.403,Z 416.201,A -85,B 0,C 180,E1 -783.636,E2 -783.636} C_VEL
LIN {X 0,Y 601.426,Z 416.227,A -85,B 0,C 180,E1 -784.521,E2 -784.521} C_VEL
LIN {X 0,Y 601.878,Z 419.738,A -85,B 0,C 180,E1 -784.958,E2 -784.958} C_VEL
LIN {X 0,Y 601.769,Z 443.189,A -85,B 0,C 180,E1 -787.698,E2 -787.698} C_VEL
LIN {X 0,Y 601.668,Z 468.118,A -85,B 0,C 180,E1 -790.555,E2 -790.555} C_VEL
LIN {X 0,Y 601.633,Z 474.862,A -85,B 0,C 180,E1 -791.319,E2 -791.319} C_VEL
LIN {X 0,Y 602.032,Z 478.967,A -85,B 0,C 180,E1 -791.388,E2 -791.388} C_VEL
LIN {X 0,Y 601.875,Z 641.56,A -85,B 0,C 180,E1 -793.398,E2 -793.398} C_VEL
LIN {X 0,Y 601.813,Z 657.481,A -85,B 0,C 180,E1 -793.745,E2 -793.745} C_VEL
LIN {X 0,Y 601.765,Z 672.043,A -85,B 0,C 180,E1 -794.201,E2 -794.201} C_VEL
LIN {X 0,Y 601.719,Z 685.754,A -85,B 0,C 180,E1 -794.764,E2 -794.764} C_VEL
LIN {X 0,Y 601.658,Z 699.229,A -85,B 0,C 180,E1 -795.455,E2 -795.455} C_VEL
LIN {X 0,Y 601.617,Z 712.447,A -85,B 0,C 180,E1 -796.283,E2 -796.283} C_VEL
LIN {X 0,Y 601.531,Z 724.281,A -85,B 0,C 180,E1 -797.174,E2 -797.174} C_VEL
LIN {X 0,Y 601.488,Z 735.745,A -85,B 0,C 180,E1 -798.201,E2 -798.201} C_VEL
LIN {X 0,Y 601.43,Z 745.386,A -85,B 0,C 180,E1 -799.224,E2 -799.224} C_VEL
LIN {X 0,Y 601.428,Z 754.852,A -85,B 0,C 180,E1 -800.414,E2 -800.414} C_VEL
LIN {X 0,Y 601.368,Z 762.728,A -85,B 0,C 180,E1 -801.6,E2 -801.6} C_VEL
LIN {X 0,Y 601.369,Z 770.086,A -85,B 0,C 180,E1 -802.951,E2 -802.951} C_VEL
LIN {X 0,Y 601.371,Z 775.923,A -85,B 0,C 180,E1 -804.299,E2 -804.299} C_VEL
LIN {X 0,Y 601.33,Z 779.382,A -85,B 0,C 180,E1 -805.307,E2 -805.307} C_VEL
LIN {X 0,Y 601.337,Z 782.885,A -85,B 0,C 180,E1 -806.65,E2 -806.65} C_VEL
LIN {X 0,Y 601.339,Z 785.191,A -85,B 0,C 180,E1 -807.99,E2 -807.99} C_VEL
LIN {X 0,Y 601.337,Z 786.35,A -85,B 0,C 180,E1 -809.33,E2 -809.33} C_VEL
LIN {X 0,Y 601.336,Z 786.35,A -85,B 0,C 180,E1 -810.669,E2 -810.669} C_VEL
LIN {X 0,Y 601.339,Z 785.192,A -85,B 0,C 180,E1 -812.009,E2 -812.009} C_VEL
LIN {X 0,Y 601.337,Z 782.887,A -85,B 0,C 180,E1 -813.35,E2 -813.35} C_VEL
LIN {X 0,Y 601.33,Z 779.384,A -85,B 0,C 180,E1 -814.692,E2 -814.692} C_VEL
LIN {X 0,Y 601.352,Z 774.61,A -85,B 0,C 180,E1 -816.037,E2 -816.037} C_VEL
LIN {X 0,Y 601.382,Z 768.428,A -85,B 0,C 180,E1 -817.385,E2 -817.385} C_VEL
LIN {X 0,Y 601.387,Z 760.656,A -85,B 0,C 180,E1 -818.738,E2 -818.738} C_VEL
LIN {X 0,Y 601.427,Z 752.374,A -85,B 0,C 180,E1 -819.925,E2 -819.925} C_VEL
LIN {X 0,Y 601.46,Z 741.935,A -85,B 0,C 180,E1 -821.164,E2 -821.164} C_VEL
LIN {X 0,Y 601.513,Z 732.198,A -85,B 0,C 180,E1 -822.14,E2 -822.14} C_VEL
LIN {X 0,Y 601.57,Z 720.022,A -85,B 0,C 180,E1 -823.168,E2 -823.168} C_VEL
LIN {X 0,Y 601.605,Z 708.085,A -85,B 0,C 180,E1 -824.011,E2 -824.011} C_VEL
LIN {X 0,Y 601.65,Z 694.537,A -85,B 0,C 180,E1 -824.804,E2 -824.804} C_VEL
LIN {X 0,Y 601.761,Z 679.856,A -85,B 0,C 180,E1 -825.495,E2 -825.495} C_VEL
LIN {X 0,Y 601.782,Z 665.635,A -85,B 0,C 180,E1 -826.016,E2 -826.016} C_VEL
LIN {X 0,Y 601.856,Z 650.707,A -85,B 0,C 180,E1 -826.42,E2 -826.42} C_VEL
LIN {X 0,Y 601.867,Z 635.741,A -85,B 0,C 180,E1 -826.689,E2 -826.689} C_VEL
LIN {X 0,Y 601.909,Z 476.419,A -85,B 0,C 180,E1 -828.648,E2 -828.648} C_VEL
LIN {X 0,Y 601.654,Z 474.74,A -85,B 0,C 180,E1 -828.695,E2 -828.695} C_VEL
LIN {X 0,Y 601.74,Z 449.397,A -85,B 0,C 180,E1 -831.586,E2 -831.586} C_VEL
LIN {X 0,Y 601.878,Z 425.303,A -85,B 0,C 180,E1 -834.386,E2 -834.386} C_VEL
LIN {X 0,Y 601.85,Z 418.184,A -85,B 0,C 180,E1 -835.227,E2 -835.227} C_VEL
LIN {X 0,Y 601.421,Z 416.194,A -85,B 0,C 180,E1 -835.501,E2 -835.501} C_VEL
LIN {X 0,Y 601.42,Z 416.194,A -85,B 0,C 180,E1 -837.867,E2 -837.867} C_VEL
LIN {X 0,Y 601.426,Z 416.197,A -85,B 0,C 180,E1 -840.163,E2 -840.163} C_VEL
LIN {X 0,Y 601.422,Z 416.192,A -85,B 0,C 180,E1 -842.716,E2 -842.716} C_VEL
LIN {X 0,Y 601.392,Z 416.192,A -85,B 0,C 180,E1 -845.111,E2 -845.111} C_VEL
LIN {X 0,Y 601.433,Z 416.187,A -85,B 0,C 180,E1 -847.418,E2 -847.418} C_VEL
LIN {X 0,Y 601.409,Z 416.195,A -85,B 0,C 180,E1 -849.994,E2 -849.994} C_VEL
LIN {X 0,Y 601.434,Z 416.191,A -85,B 0,C 180,E1 -852.667,E2 -852.667} C_VEL
LIN {X 0,Y 601.42,Z 416.189,A -85,B 0,C 180,E1 -855.482,E2 -855.482} C_VEL
LIN {X 0,Y 601.419,Z 416.198,A -85,B 0,C 180,E1 -858.406,E2 -858.406} C_VEL
LIN {X 0,Y 601.432,Z 416.189,A -85,B 0,C 180,E1 -860.875,E2 -860.875} C_VEL
LIN {X 0,Y 601.437,Z 416.188,A -85,B 0,C 180,E1 -863.733,E2 -863.733} C_VEL
LIN {X 0,Y 601.429,Z 416.193,A -85,B 0,C 180,E1 -866.063,E2 -866.063} C_VEL
LIN {X 0,Y 601.435,Z 416.193,A -85,B 0,C 180,E1 -868.541,E2 -868.541} C_VEL
LIN {X 0,Y 601.431,Z 416.187,A -85,B 0,C 180,E1 -871.373,E2 -871.373} C_VEL
LIN {X 0,Y 601.417,Z 416.196,A -85,B 0,C 180,E1 -874.13,E2 -874.13} C_VEL
LIN {X 0,Y 601.416,Z 416.195,A -85,B 0,C 180,E1 -876.59,E2 -876.59} C_VEL
LIN {X 0,Y 601.429,Z 416.187,A -85,B 0,C 180,E1 -879.478,E2 -879.478} C_VEL
LIN {X 0,Y 601.392,Z 416.202,A -85,B 0,C 180,E1 -882.312,E2 -882.312} C_VEL
LIN {X 0,Y 601.41,Z 416.199,A -85,B 0,C 180,E1 -884.409,E2 -884.409} C_VEL
LIN {X 0,Y 601.419,Z 416.188,A -85,B 0,C 180,E1 -887.172,E2 -887.172} C_VEL
LIN {X 0,Y 601.433,Z 416.19,A -85,B 0,C 180,E1 -889.905,E2 -889.905} C_VEL
LIN {X 0,Y 601.435,Z 416.193,A -85,B 0,C 180,E1 -892.615,E2 -892.615} C_VEL
LIN {X 0,Y 601.429,Z 416.187,A -85,B 0,C 180,E1 -895.308,E2 -895.308} C_VEL
LIN {X 0,Y 601.423,Z 416.192,A -85,B 0,C 180,E1 -897.991,E2 -897.991} C_VEL
LIN {X 0,Y 601.448,Z 416.19,A -85,B 0,C 180,E1 -900.67,E2 -900.67} C_VEL
LIN {X 0,Y 601.427,Z 416.187,A -85,B 0,C 180,E1 -903.35,E2 -903.35} C_VEL
LIN {X 0,Y 601.431,Z 416.191,A -85,B 0,C 180,E1 -906.037,E2 -906.037} C_VEL
LIN {X 0,Y 601.437,Z 416.191,A -85,B 0,C 180,E1 -908.738,E2 -908.738} C_VEL
LIN {X 0,Y 601.429,Z 416.187,A -85,B 0,C 180,E1 -911.458,E2 -911.458} C_VEL
LIN {X 0,Y 601.409,Z 416.193,A -85,B 0,C 180,E1 -912.386,E2 -912.386} C_VEL
LIN {X 0,Y 600.745,Z 416.275,A -85,B 0,C 180,E1 -912.946,E2 -912.946} C_VEL
LIN {X 0,Y 597.894,Z 416.63,A -85,B 0,C 180,E1 -913.854,E2 -913.854} C_VEL
LIN {X 0,Y 595.482,Z 416.936,A -85,B 0,C 180,E1 -914.584,E2 -914.584} C_VEL
LIN {X 0,Y 594.444,Z 417.059,A -85,B 0,C 180,E1 -915.147,E2 -915.147} C_VEL
LIN {X 0,Y 594.359,Z 417.068,A -85,B 0,C 180,E1 -915.338,E2 -915.338} C_VEL
LIN {X 0,Y 594.376,Z 417.068,A -85,B 0,C 180,E1 -917.905,E2 -917.905} C_VEL
LIN {X 0,Y 594.38,Z 417.068,A -85,B 0,C 180,E1 -920.919,E2 -920.919} C_VEL
LIN {X 0,Y 594.389,Z 417.065,A -85,B 0,C 180,E1 -923.704,E2 -923.704} C_VEL
LIN {X 0,Y 594.383,Z 417.071,A -85,B 0,C 180,E1 -926.7,E2 -926.7} C_VEL
LIN {X 0,Y 594.383,Z 417.067,A -85,B 0,C 180,E1 -928.999,E2 -928.999} C_VEL
LIN {X 0,Y 594.39,Z 417.065,A -85,B 0,C 180,E1 -931.646,E2 -931.646} C_VEL
LIN {X 0,Y 594.395,Z 417.072,A -85,B 0,C 180,E1 -934.579,E2 -934.579} C_VEL
LIN {X 0,Y 594.381,Z 417.067,A -85,B 0,C 180,E1 -937.087,E2 -937.087} C_VEL
LIN {X 0,Y 594.376,Z 417.068,A -85,B 0,C 180,E1 -939.776,E2 -939.776} C_VEL
LIN {X 0,Y 594.367,Z 417.077,A -85,B 0,C 180,E1 -942.376,E2 -942.376} C_VEL
LIN {X 0,Y 594.395,Z 417.111,A -85,B 0,C 180,E1 -945.275,E2 -945.275} C_VEL
LIN {X 0,Y 594.79,Z 420.882,A -85,B 0,C 180,E1 -945.803,E2 -945.803} C_VEL
LIN {X 0,Y 594.659,Z 442.72,A -85,B 0,C 180,E1 -948.728,E2 -948.728} C_VEL
LIN {X 0,Y 594.636,Z 445.904,A -85,B 0,C 180,E1 -949.15,E2 -949.15} C_VEL
LIN {X 0,Y 595.31,Z 450.186,A -85,B 0,C 180,E1 -949.23,E2 -949.23} C_VEL
LIN {X 0,Y 595.095,Z 610.993,A -85,B 0,C 180,E1 -951.238,E2 -951.238} C_VEL
LIN {X 0,Y 594.981,Z 626.865,A -85,B 0,C 180,E1 -951.58,E2 -951.58} C_VEL
LIN {X 0,Y 594.949,Z 641.749,A -85,B 0,C 180,E1 -952.049,E2 -952.049} C_VEL
LIN {X 0,Y 594.847,Z 656.329,A -85,B 0,C 180,E1 -952.654,E2 -952.654} C_VEL
LIN {X 0,Y 594.752,Z 670.572,A -85,B 0,C 180,E1 -953.402,E2 -953.402} C_VEL
LIN {X 0,Y 594.62,Z 684.385,A -85,B 0,C 180,E1 -954.298,E2 -954.298} C_VEL
LIN {X 0,Y 594.53,Z 696.223,A -85,B 0,C 180,E1 -955.225,E2 -955.225} C_VEL
LIN {X 0,Y 594.473,Z 707.192,A -85,B 0,C 180,E1 -956.246,E2 -956.246} C_VEL
LIN {X 0,Y 594.394,Z 718.061,A -85,B 0,C 180,E1 -957.454,E2 -957.454} C_VEL
LIN {X 0,Y 594.353,Z 727.037,A -85,B 0,C 180,E1 -958.65,E2 -958.65} C_VEL
LIN {X 0,Y 594.313,Z 735.129,A -85,B 0,C 180,E1 -959.952,E2 -959.952} C_VEL
LIN {X 0,Y 594.259,Z 740.811,A -85,B 0,C 180,E1 -961.065,E2 -961.065} C_VEL
LIN {X 0,Y 594.268,Z 746.725,A -85,B 0,C 180,E1 -962.496,E2 -962.496} C_VEL
LIN {X 0,Y 594.274,Z 749.382,A -85,B 0,C 180,E1 -963.296,E2 -963.296} C_VEL
LIN {X 0,Y 594.219,Z 753.194,A -85,B 0,C 180,E1 -964.801,E2 -964.801} C_VEL
LIN {X 0,Y 594.223,Z 755.512,A -85,B 0,C 180,E1 -966.29,E2 -966.29} C_VEL
LIN {X 0,Y 594.251,Z 756.441,A -85,B 0,C 180,E1 -967.763,E2 -967.763} C_VEL
LIN {X 0,Y 594.25,Z 756.037,A -85,B 0,C 180,E1 -969.219,E2 -969.219} C_VEL
LIN {X 0,Y 594.21,Z 754.342,A -85,B 0,C 180,E1 -970.661,E2 -970.661} C_VEL
LIN {X 0,Y 594.21,Z 751.349,A -85,B 0,C 180,E1 -972.091,E2 -972.091} C_VEL
LIN {X 0,Y 594.252,Z 747.026,A -85,B 0,C 180,E1 -973.511,E2 -973.511} C_VEL
LIN {X 0,Y 594.29,Z 741.307,A -85,B 0,C 180,E1 -974.92,E2 -974.92} C_VEL
LIN {X 0,Y 594.296,Z 734.067,A -85,B 0,C 180,E1 -976.32,E2 -976.32} C_VEL
LIN {X 0,Y 594.353,Z 726.348,A -85,B 0,C 180,E1 -977.538,E2 -977.538} C_VEL
LIN {X 0,Y 594.417,Z 716.978,A -85,B 0,C 180,E1 -978.765,E2 -978.765} C_VEL
LIN {X 0,Y 594.464,Z 707.761,A -85,B 0,C 180,E1 -979.786,E2 -979.786} C_VEL
LIN {X 0,Y 594.545,Z 695.755,A -85,B 0,C 180,E1 -980.904,E2 -980.904} C_VEL
LIN {X 0,Y 594.648,Z 683.603,A -85,B 0,C 180,E1 -981.847,E2 -981.847} C_VEL
LIN {X 0,Y 594.75,Z 670.313,A -85,B 0,C 180,E1 -982.703,E2 -982.703} C_VEL
LIN {X 0,Y 594.843,Z 655.802,A -85,B 0,C 180,E1 -983.46,E2 -983.46} C_VEL
LIN {X 0,Y 594.952,Z 640.975,A -85,B 0,C 180,E1 -984.068,E2 -984.068} C_VEL
LIN {X 0,Y 595.041,Z 625.75,A -85,B 0,C 180,E1 -984.536,E2 -984.536} C_VEL
LIN {X 0,Y 595.08,Z 610.852,A -85,B 0,C 180,E1 -984.855,E2 -984.855} C_VEL
LIN {X 0,Y 595.198,Z 448.841,A -85,B 0,C 180,E1 -986.88,E2 -986.88} C_VEL
LIN {X 0,Y 594.624,Z 445.822,A -85,B 0,C 180,E1 -986.952,E2 -986.952} C_VEL
LIN {X 0,Y 594.767,Z 425.512,A -85,B 0,C 180,E1 -989.662,E2 -989.662} C_VEL
LIN {X 0,Y 594.574,Z 418.065,A -85,B 0,C 180,E1 -990.678,E2 -990.678} C_VEL
LIN {X 0,Y 594.409,Z 417.068,A -85,B 0,C 180,E1 -990.847,E2 -990.847} C_VEL
LIN {X 0,Y 594.388,Z 417.072,A -85,B 0,C 180,E1 -993.39,E2 -993.39} C_VEL
LIN {X 0,Y 594.368,Z 417.07,A -85,B 0,C 180,E1 -996.109,E2 -996.109} C_VEL
LIN {X 0,Y 594.381,Z 417.066,A -85,B 0,C 180,E1 -998.842,E2 -998.842} C_VEL
LIN {X 0,Y 594.4,Z 417.072,A -85,B 0,C 180,E1 -1001.596,E2 -1001.596} C_VEL
LIN {X 0,Y 594.394,Z 417.064,A -85,B 0,C 180,E1 -1004.377,E2 -1004.377} C_VEL
LIN {X 0,Y 594.385,Z 417.068,A -85,B 0,C 180,E1 -1007.194,E2 -1007.194} C_VEL
LIN {X 0,Y 594.379,Z 417.069,A -85,B 0,C 180,E1 -1010.054,E2 -1010.054} C_VEL
LIN {X 0,Y 594.369,Z 417.068,A -85,B 0,C 180,E1 -1012.967,E2 -1012.967} C_VEL
LIN {X 0,Y 594.381,Z 417.068,A -85,B 0,C 180,E1 -1015.193,E2 -1015.193} C_VEL
LIN {X 0,Y 594.39,Z 417.073,A -85,B 0,C 180,E1 -1017.527,E2 -1017.527} C_VEL
LIN {X 0,Y 594.392,Z 417.065,A -85,B 0,C 180,E1 -1020.328,E2 -1020.328} C_VEL
LIN {X 0,Y 594.381,Z 417.065,A -85,B 0,C 180,E1 -1022.95,E2 -1022.95} C_VEL
LIN {X 0,Y 594.359,Z 417.074,A -85,B 0,C 180,E1 -1025.408,E2 -1025.408} C_VEL
LIN {X 0,Y 594.391,Z 417.069,A -85,B 0,C 180,E1 -1027.94,E2 -1027.94} C_VEL
LIN {X 0,Y 594.38,Z 417.065,A -85,B 0,C 180,E1 -1030.822,E2 -1030.822} C_VEL
LIN {X 0,Y 594.385,Z 417.072,A -85,B 0,C 180,E1 -1033.841,E2 -1033.841} C_VEL
LIN {X 0,Y 594.368,Z 417.067,A -85,B 0,C 180,E1 -1036.7,E2 -1036.7} C_VEL
LIN {X 0,Y 594.374,Z 417.072,A -85,B 0,C 180,E1 -1039.433,E2 -1039.433} C_VEL
LIN {X 0,Y 594.39,Z 417.064,A -85,B 0,C 180,E1 -1042.391,E2 -1042.391} C_VEL
LIN {X 0,Y 594.386,Z 417.064,A -85,B 0,C 180,E1 -1044.671,E2 -1044.671} C_VEL
LIN {X 0,Y 594.38,Z 417.067,A -85,B 0,C 180,E1 -1047.088,E2 -1047.088} C_VEL
LIN {X 0,Y 594.387,Z 417.074,A -85,B 0,C 180,E1 -1049.671,E2 -1049.671} C_VEL
LIN {X 0,Y 594.375,Z 417.066,A -85,B 0,C 180,E1 -1052.539,E2 -1052.539} C_VEL
LIN {X 0,Y 594.378,Z 417.065,A -85,B 0,C 180,E1 -1054.807,E2 -1054.807} C_VEL
LIN {X 0,Y 594.365,Z 417.07,A -85,B 0,C 180,E1 -1057.264,E2 -1057.264} C_VEL
LIN {X 0,Y 594.377,Z 417.071,A -85,B 0,C 180,E1 -1059.946,E2 -1059.946} C_VEL
LIN {X 0,Y 594.39,Z 417.063,A -85,B 0,C 180,E1 -1062.806,E2 -1062.806} C_VEL
LIN {X 0,Y 594.389,Z 417.072,A -85,B 0,C 180,E1 -1065.826,E2 -1065.826} C_VEL
LIN {X 0,Y 594.393,Z 417.064,A -85,B 0,C 180,E1 -1068.404,E2 -1068.404} C_VEL
LIN {X 0,Y 594.399,Z 417.064,A -85,B 0,C 180,E1 -1071.158,E2 -1071.158} C_VEL
LIN {X 0,Y 594.37,Z 417.073,A -85,B 0,C 180,E1 -1073.891,E2 -1073.891} C_VEL
LIN {X 0,Y 594.379,Z 417.064,A -85,B 0,C 180,E1 -1076.61,E2 -1076.61} C_VEL
LIN {X 0,Y 594.42,Z 417.064,A -85,B 0,C 180,E1 -1079.322,E2 -1079.322} C_VEL
LIN {X 0,Y 594.396,Z 417.068,A -85,B 0,C 180,E1 -1082.033,E2 -1082.033} C_VEL
LIN {X 0,Y 594.397,Z 417.061,A -85,B 0,C 180,E1 -1084.747,E2 -1084.747} C_VEL
LIN {X 0,Y 594.392,Z 417.07,A -85,B 0,C 180,E1 -1087.473,E2 -1087.473} C_VEL
LIN {X 0,Y 594.395,Z 417.065,A -85,B 0,C 180,E1 -1090.216,E2 -1090.216} C_VEL
LIN {X 0,Y 594.367,Z 417.067,A -85,B 0,C 180,E1 -1092.983,E2 -1092.983} C_VEL
LIN {X 0,Y 594.366,Z 417.076,A -85,B 0,C 180,E1 -1095.781,E2 -1095.781} C_VEL
LIN {X 0,Y 594.387,Z 417.063,A -85,B 0,C 180,E1 -1098.617,E2 -1098.617} C_VEL
LIN {X 0,Y 594.366,Z 417.074,A -85,B 0,C 180,E1 -1101.503,E2 -1101.503} C_VEL
LIN {X 0,Y 594.387,Z 417.065,A -85,B 0,C 180,E1 -1104.446,E2 -1104.446} C_VEL
LIN {X 0,Y 594.382,Z 417.065,A -85,B 0,C 180,E1 -1106.7,E2 -1106.7} C_VEL
LIN {X 0,Y 594.381,Z 417.066,A -85,B 0,C 180,E1 -1108.998,E2 -1108.998} C_VEL
LIN {X 0,Y 594.376,Z 417.075,A -85,B 0,C 180,E1 -1111.643,E2 -1111.643} C_VEL
LIN {X 0,Y 594.395,Z 417.063,A -85,B 0,C 180,E1 -1114.579,E2 -1114.579} C_VEL
LIN {X 0,Y 594.384,Z 417.066,A -85,B 0,C 180,E1 -1117.087,E2 -1117.087} C_VEL
LIN {X 0,Y 594.376,Z 417.076,A -85,B 0,C 180,E1 -1119.775,E2 -1119.775} C_VEL
LIN {X 0,Y 594.365,Z 417.068,A -85,B 0,C 180,E1 -1122.376,E2 -1122.376} C_VEL
LIN {X 0,Y 594.363,Z 417.07,A -85,B 0,C 180,E1 -1125.191,E2 -1125.191} C_VEL
LIN {X 0,Y 594.371,Z 417.076,A -85,B 0,C 180,E1 -1127.625,E2 -1127.625} C_VEL
LIN {X 0,Y 594.373,Z 417.068,A -85,B 0,C 180,E1 -1130.319,E2 -1130.319} C_VEL
LIN {X 0,Y 594.383,Z 417.065,A -85,B 0,C 180,E1 -1132.913,E2 -1132.913} C_VEL
LIN {X 0,Y 594.381,Z 417.074,A -85,B 0,C 180,E1 -1135.861,E2 -1135.861} C_VEL
LIN {X 0,Y 594.381,Z 417.066,A -85,B 0,C 180,E1 -1138.65,E2 -1138.65} C_VEL
LIN {X 0,Y 594.383,Z 417.067,A -85,B 0,C 180,E1 -1141.042,E2 -1141.042} C_VEL
LIN {X 0,Y 594.383,Z 417.075,A -85,B 0,C 180,E1 -1143.978,E2 -1143.978} C_VEL
LIN {X 0,Y 594.394,Z 417.202,A -85,B 0,C 180,E1 -1144.315,E2 -1144.315} C_VEL
LIN {X 0,Y 595.088,Z 421.299,A -85,B 0,C 180,E1 -1144.839,E2 -1144.839} C_VEL
LIN {X 0,Y 594.91,Z 444.939,A -85,B 0,C 180,E1 -1147.632,E2 -1147.632} C_VEL
LIN {X 0,Y 594.759,Z 469.679,A -85,B 0,C 180,E1 -1150.499,E2 -1150.499} C_VEL
LIN {X 0,Y 594.704,Z 474.88,A -85,B 0,C 180,E1 -1151.095,E2 -1151.095} C_VEL
LIN {X 0,Y 595.313,Z 478.419,A -85,B 0,C 180,E1 -1151.163,E2 -1151.163} C_VEL
LIN {X 0,Y 595.083,Z 641.353,A -85,B 0,C 180,E1 -1153.199,E2 -1153.199} C_VEL
LIN {X 0,Y 595.017,Z 656.703,A -85,B 0,C 180,E1 -1153.532,E2 -1153.532} C_VEL
LIN {X 0,Y 594.931,Z 672.042,A -85,B 0,C 180,E1 -1154.014,E2 -1154.014} C_VEL
LIN {X 0,Y 594.857,Z 685.757,A -85,B 0,C 180,E1 -1154.584,E2 -1154.584} C_VEL
LIN {X 0,Y 594.732,Z 699.231,A -85,B 0,C 180,E1 -1155.281,E2 -1155.281} C_VEL
LIN {X 0,Y 594.681,Z 711.789,A -85,B 0,C 180,E1 -1156.075,E2 -1156.075} C_VEL
LIN {X 0,Y 594.56,Z 724.283,A -85,B 0,C 180,E1 -1157.021,E2 -1157.021} C_VEL
LIN {X 0,Y 594.465,Z 735.746,A -85,B 0,C 180,E1 -1158.059,E2 -1158.059} C_VEL
LIN {X 0,Y 594.388,Z 745.387,A -85,B 0,C 180,E1 -1159.095,E2 -1159.095} C_VEL
LIN {X 0,Y 594.366,Z 754.853,A -85,B 0,C 180,E1 -1160.299,E2 -1160.299} C_VEL
LIN {X 0,Y 594.311,Z 762.729,A -85,B 0,C 180,E1 -1161.499,E2 -1161.499} C_VEL
LIN {X 0,Y 594.293,Z 770.087,A -85,B 0,C 180,E1 -1162.867,E2 -1162.867} C_VEL
LIN {X 0,Y 594.296,Z 775.923,A -85,B 0,C 180,E1 -1164.231,E2 -1164.231} C_VEL
LIN {X 0,Y 594.232,Z 779.383,A -85,B 0,C 180,E1 -1165.251,E2 -1165.251} C_VEL
LIN {X 0,Y 594.257,Z 782.886,A -85,B 0,C 180,E1 -1166.61,E2 -1166.61} C_VEL
LIN {X 0,Y 594.238,Z 785.192,A -85,B 0,C 180,E1 -1167.966,E2 -1167.966} C_VEL
LIN {X 0,Y 594.237,Z 786.35,A -85,B 0,C 180,E1 -1169.322,E2 -1169.322} C_VEL
LIN {X 0,Y 594.237,Z 786.35,A -85,B 0,C 180,E1 -1170.677,E2 -1170.677} C_VEL
LIN {X 0,Y 594.238,Z 785.193,A -85,B 0,C 180,E1 -1172.033,E2 -1172.033} C_VEL
LIN {X 0,Y 594.257,Z 782.887,A -85,B 0,C 180,E1 -1173.39,E2 -1173.39} C_VEL
LIN {X 0,Y 594.232,Z 779.385,A -85,B 0,C 180,E1 -1174.748,E2 -1174.748} C_VEL
LIN {X 0,Y 594.275,Z 774.61,A -85,B 0,C 180,E1 -1176.109,E2 -1176.109} C_VEL
LIN {X 0,Y 594.296,Z 768.427,A -85,B 0,C 180,E1 -1177.474,E2 -1177.474} C_VEL
LIN {X 0,Y 594.331,Z 760.655,A -85,B 0,C 180,E1 -1178.842,E2 -1178.842} C_VEL
LIN {X 0,Y 594.387,Z 752.374,A -85,B 0,C 180,E1 -1180.043,E2 -1180.043} C_VEL
LIN {X 0,Y 594.433,Z 742.561,A -85,B 0,C 180,E1 -1181.231,E2 -1181.231} C_VEL
LIN {X 0,Y 594.53,Z 732.197,A -85,B 0,C 180,E1 -1182.285,E2 -1182.285} C_VEL
LIN {X 0,Y 594.581,Z 720.023,A -85,B 0,C 180,E1 -1183.325,E2 -1183.325} C_VEL
LIN {X 0,Y 594.693,Z 708.083,A -85,B 0,C 180,E1 -1184.177,E2 -1184.177} C_VEL
LIN {X 0,Y 594.75,Z 694.535,A -85,B 0,C 180,E1 -1184.98,E2 -1184.98} C_VEL
LIN {X 0,Y 594.902,Z 679.853,A -85,B 0,C 180,E1 -1185.678,E2 -1185.678} C_VEL
LIN {X 0,Y 594.951,Z 665.634,A -85,B 0,C 180,E1 -1186.204,E2 -1186.204} C_VEL
LIN {X 0,Y 595.048,Z 651.139,A -85,B 0,C 180,E1 -1186.602,E2 -1186.602} C_VEL
LIN {X 0,Y 595.067,Z 635.741,A -85,B 0,C 180,E1 -1186.886,E2 -1186.886} C_VEL
LIN {X 0,Y 595.211,Z 477.72,A -85,B 0,C 180,E1 -1188.849,E2 -1188.849} C_VEL
LIN {X 0,Y 594.732,Z 474.801,A -85,B 0,C 180,E1 -1188.913,E2 -1188.913} C_VEL
LIN {X 0,Y 594.88,Z 450.958,A -85,B 0,C 180,E1 -1191.665,E2 -1191.665} C_VEL
LIN {X 0,Y 595.056,Z 427.548,A -85,B 0,C 180,E1 -1194.416,E2 -1194.416} C_VEL
LIN {X 0,Y 594.983,Z 419.745,A -85,B 0,C 180,E1 -1195.352,E2 -1195.352} C_VEL
LIN {X 0,Y 594.384,Z 417.073,A -85,B 0,C 180,E1 -1195.708,E2 -1195.708} C_VEL
LIN {X 0,Y 594.383,Z 417.077,A -85,B 0,C 180,E1 -1198.226,E2 -1198.226} C_VEL
LIN {X 0,Y 594.386,Z 417.071,A -85,B 0,C 180,E1 -1200.558,E2 -1200.558} C_VEL
LIN {X 0,Y 594.376,Z 417.067,A -85,B 0,C 180,E1 -1202.949,E2 -1202.949} C_VEL
LIN {X 0,Y 594.351,Z 417.069,A -85,B 0,C 180,E1 -1205.408,E2 -1205.408} C_VEL
LIN {X 0,Y 594.386,Z 417.069,A -85,B 0,C 180,E1 -1207.94,E2 -1207.94} C_VEL
LIN {X 0,Y 594.377,Z 417.068,A -85,B 0,C 180,E1 -1210.822,E2 -1210.822} C_VEL
LIN {X 0,Y 594.382,Z 417.065,A -85,B 0,C 180,E1 -1213.297,E2 -1213.297} C_VEL
LIN {X 0,Y 594.362,Z 417.076,A -85,B 0,C 180,E1 -1216.16,E2 -1216.16} C_VEL
LIN {X 0,Y 594.376,Z 417.073,A -85,B 0,C 180,E1 -1218.536,E2 -1218.536} C_VEL
LIN {X 0,Y 594.382,Z 417.065,A -85,B 0,C 180,E1 -1221.295,E2 -1221.295} C_VEL
LIN {X 0,Y 594.39,Z 417.066,A -85,B 0,C 180,E1 -1223.758,E2 -1223.758} C_VEL
LIN {X 0,Y 594.375,Z 417.075,A -85,B 0,C 180,E1 -1226.239,E2 -1226.239} C_VEL
LIN {X 0,Y 594.384,Z 417.07,A -85,B 0,C 180,E1 -1228.651,E2 -1228.651} C_VEL
LIN {X 0,Y 594.38,Z 417.066,A -85,B 0,C 180,E1 -1231.041,E2 -1231.041} C_VEL
LIN {X 0,Y 594.389,Z 417.068,A -85,B 0,C 180,E1 -1233.975,E2 -1233.975} C_VEL
LIN {X 0,Y 594.385,Z 417.075,A -85,B 0,C 180,E1 -1236.296,E2 -1236.296} C_VEL
LIN {X 0,Y 594.401,Z 417.062,A -85,B 0,C 180,E1 -1239.224,E2 -1239.224} C_VEL
LIN {X 0,Y 594.374,Z 417.072,A -85,B 0,C 180,E1 -1242.096,E2 -1242.096} C_VEL
LIN {X 0,Y 594.364,Z 417.075,A -85,B 0,C 180,E1 -1244.219,E2 -1244.219} C_VEL
LIN {X 0,Y 594.365,Z 417.068,A -85,B 0,C 180,E1 -1247.017,E2 -1247.017} C_VEL
LIN {X 0,Y 594.392,Z 417.066,A -85,B 0,C 180,E1 -1249.784,E2 -1249.784} C_VEL
LIN {X 0,Y 594.388,Z 417.072,A -85,B 0,C 180,E1 -1252.527,E2 -1252.527} C_VEL
LIN {X 0,Y 594.396,Z 417.063,A -85,B 0,C 180,E1 -1255.253,E2 -1255.253} C_VEL
LIN {X 0,Y 594.393,Z 417.067,A -85,B 0,C 180,E1 -1257.967,E2 -1257.967} C_VEL
LIN {X 0,Y 594.419,Z 417.065,A -85,B 0,C 180,E1 -1260.678,E2 -1260.678} C_VEL
LIN {X 0,Y 594.378,Z 417.065,A -85,B 0,C 180,E1 -1263.39,E2 -1263.39} C_VEL
LIN {X 0,Y 594.384,Z 417.07,A -85,B 0,C 180,E1 -1266.109,E2 -1266.109} C_VEL
LIN {X 0,Y 594.396,Z 417.067,A -85,B 0,C 180,E1 -1268.842,E2 -1268.842} C_VEL
LIN {X 0,Y 594.389,Z 417.064,A -85,B 0,C 180,E1 -1271.596,E2 -1271.596} C_VEL
LIN {X 0,Y 594.384,Z 417.075,A -85,B 0,C 180,E1 -1274.377,E2 -1274.377} C_VEL
LIN {X 0,Y 594.359,Z 417.068,A -85,B 0,C 180,E1 -1275.338,E2 -1275.338} C_VEL
LIN {X 0,Y 593.689,Z 417.155,A -85,B 0,C 180,E1 -1275.904,E2 -1275.904} C_VEL
LIN {X 0,Y 590.835,Z 417.511,A -85,B 0,C 180,E1 -1276.822,E2 -1276.822} C_VEL
LIN {X 0,Y 588.43,Z 417.813,A -85,B 0,C 180,E1 -1277.561,E2 -1277.561} C_VEL
LIN {X 0,Y 587.403,Z 417.94,A -85,B 0,C 180,E1 -1278.131,E2 -1278.131} C_VEL
LIN {X 0,Y 587.322,Z 417.948,A -85,B 0,C 180,E1 -1278.324,E2 -1278.324} C_VEL
LIN {X 0,Y 587.352,Z 417.942,A -85,B 0,C 180,E1 -1281.045,E2 -1281.045} C_VEL
LIN {X 0,Y 587.334,Z 417.947,A -85,B 0,C 180,E1 -1284.007,E2 -1284.007} C_VEL
LIN {X 0,Y 587.36,Z 417.948,A -85,B 0,C 180,E1 -1286.278,E2 -1286.278} C_VEL
LIN {X 0,Y 587.35,Z 417.942,A -85,B 0,C 180,E1 -1289.135,E2 -1289.135} C_VEL
LIN {X 0,Y 587.354,Z 417.943,A -85,B 0,C 180,E1 -1291.839,E2 -1291.839} C_VEL
LIN {X 0,Y 587.354,Z 417.95,A -85,B 0,C 180,E1 -1294.35,E2 -1294.35} C_VEL
LIN {X 0,Y 587.349,Z 417.947,A -85,B 0,C 180,E1 -1296.747,E2 -1296.747} C_VEL
LIN {X 0,Y 587.344,Z 417.943,A -85,B 0,C 180,E1 -1299.36,E2 -1299.36} C_VEL
LIN {X 0,Y 587.331,Z 417.949,A -85,B 0,C 180,E1 -1302.109,E2 -1302.109} C_VEL
LIN {X 0,Y 587.37,Z 418.037,A -85,B 0,C 180,E1 -1305.115,E2 -1305.115} C_VEL
LIN {X 0,Y 587.91,Z 421.514,A -85,B 0,C 180,E1 -1305.615,E2 -1305.615} C_VEL
LIN {X 0,Y 587.725,Z 443.9,A -85,B 0,C 180,E1 -1308.649,E2 -1308.649} C_VEL
LIN {X 0,Y 587.693,Z 445.906,A -85,B 0,C 180,E1 -1308.918,E2 -1308.918} C_VEL
LIN {X 0,Y 588.596,Z 450.61,A -85,B 0,C 180,E1 -1309.013,E2 -1309.013} C_VEL
LIN {X 0,Y 588.302,Z 610.798,A -85,B 0,C 180,E1 -1311.035,E2 -1311.035} C_VEL
LIN {X 0,Y 588.201,Z 626.455,A -85,B 0,C 180,E1 -1311.374,E2 -1311.374} C_VEL
LIN {X 0,Y 588.103,Z 641.269,A -85,B 0,C 180,E1 -1311.841,E2 -1311.841} C_VEL
LIN {X 0,Y 587.976,Z 655.692,A -85,B 0,C 180,E1 -1312.441,E2 -1312.441} C_VEL
LIN {X 0,Y 587.826,Z 669.288,A -85,B 0,C 180,E1 -1313.153,E2 -1313.153} C_VEL
LIN {X 0,Y 587.72,Z 682.861,A -85,B 0,C 180,E1 -1314.025,E2 -1314.025} C_VEL
LIN {X 0,Y 587.559,Z 696.038,A -85,B 0,C 180,E1 -1315.054,E2 -1315.054} C_VEL
LIN {X 0,Y 587.471,Z 707.146,A -85,B 0,C 180,E1 -1316.098,E2 -1316.098} C_VEL
LIN {X 0,Y 587.364,Z 717.393,A -85,B 0,C 180,E1 -1317.243,E2 -1317.243} C_VEL
LIN {X 0,Y 587.311,Z 726.307,A -85,B 0,C 180,E1 -1318.432,E2 -1318.432} C_VEL
LIN {X 0,Y 587.237,Z 734.967,A -85,B 0,C 180,E1 -1319.825,E2 -1319.825} C_VEL
LIN {X 0,Y 587.187,Z 741.594,A -85,B 0,C 180,E1 -1321.148,E2 -1321.148} C_VEL
LIN {X 0,Y 587.178,Z 747.501,A -85,B 0,C 180,E1 -1322.645,E2 -1322.645} C_VEL
LIN {X 0,Y 587.139,Z 751.126,A -85,B 0,C 180,E1 -1323.864,E2 -1323.864} C_VEL
LIN {X 0,Y 587.148,Z 754.077,A -85,B 0,C 180,E1 -1325.233,E2 -1325.233} C_VEL
LIN {X 0,Y 587.113,Z 755.954,A -85,B 0,C 180,E1 -1326.733,E2 -1326.733} C_VEL
LIN {X 0,Y 587.142,Z 756.467,A -85,B 0,C 180,E1 -1328.219,E2 -1328.219} C_VEL
LIN {X 0,Y 587.118,Z 755.665,A -85,B 0,C 180,E1 -1329.688,E2 -1329.688} C_VEL
LIN {X 0,Y 587.156,Z 753.578,A -85,B 0,C 180,E1 -1331.145,E2 -1331.145} C_VEL
LIN {X 0,Y 587.136,Z 750.186,A -85,B 0,C 180,E1 -1332.588,E2 -1332.588} C_VEL
LIN {X 0,Y 587.193,Z 745.428,A -85,B 0,C 180,E1 -1334.022,E2 -1334.022} C_VEL
LIN {X 0,Y 587.224,Z 739.247,A -85,B 0,C 180,E1 -1335.444,E2 -1335.444} C_VEL
LIN {X 0,Y 587.255,Z 731.512,A -85,B 0,C 180,E1 -1336.857,E2 -1336.857} C_VEL
LIN {X 0,Y 587.342,Z 723.249,A -85,B 0,C 180,E1 -1338.089,E2 -1338.089} C_VEL
LIN {X 0,Y 587.405,Z 713.413,A -85,B 0,C 180,E1 -1339.313,E2 -1339.313} C_VEL
LIN {X 0,Y 587.502,Z 703.411,A -85,B 0,C 180,E1 -1340.359,E2 -1340.359} C_VEL
LIN {X 0,Y 587.604,Z 691.607,A -85,B 0,C 180,E1 -1341.402,E2 -1341.402} C_VEL
LIN {X 0,Y 587.746,Z 678.626,A -85,B 0,C 180,E1 -1342.356,E2 -1342.356} C_VEL
LIN {X 0,Y 587.89,Z 665.771,A -85,B 0,C 180,E1 -1343.135,E2 -1343.135} C_VEL
LIN {X 0,Y 587.986,Z 651.798,A -85,B 0,C 180,E1 -1343.825,E2 -1343.825} C_VEL
LIN {X 0,Y 588.121,Z 637.298,A -85,B 0,C 180,E1 -1344.386,E2 -1344.386} C_VEL
LIN {X 0,Y 588.24,Z 622.306,A -85,B 0,C 180,E1 -1344.817,E2 -1344.817} C_VEL
LIN {X 0,Y 588.287,Z 606.661,A -85,B 0,C 180,E1 -1345.118,E2 -1345.118} C_VEL
LIN {X 0,Y 588.486,Z 449.824,A -85,B 0,C 180,E1 -1347.091,E2 -1347.091} C_VEL
LIN {X 0,Y 587.665,Z 445.907,A -85,B 0,C 180,E1 -1347.173,E2 -1347.173} C_VEL
LIN {X 0,Y 587.864,Z 426.241,A -85,B 0,C 180,E1 -1349.829,E2 -1349.829} C_VEL
LIN {X 0,Y 587.752,Z 420.024,A -85,B 0,C 180,E1 -1350.685,E2 -1350.685} C_VEL
LIN {X 0,Y 587.385,Z 417.944,A -85,B 0,C 180,E1 -1351.007,E2 -1351.007} C_VEL
LIN {X 0,Y 587.34,Z 417.951,A -85,B 0,C 180,E1 -1353.43,E2 -1353.43} C_VEL
LIN {X 0,Y 587.32,Z 417.948,A -85,B 0,C 180,E1 -1356.183,E2 -1356.183} C_VEL
LIN {X 0,Y 587.369,Z 417.941,A -85,B 0,C 180,E1 -1358.255,E2 -1358.255} C_VEL
LIN {X 0,Y 587.353,Z 417.943,A -85,B 0,C 180,E1 -1361.134,E2 -1361.134} C_VEL
LIN {X 0,Y 587.37,Z 417.94,A -85,B 0,C 180,E1 -1364.261,E2 -1364.261} C_VEL
LIN {X 0,Y 587.35,Z 417.948,A -85,B 0,C 180,E1 -1367.406,E2 -1367.406} C_VEL
LIN {X 0,Y 587.331,Z 417.945,A -85,B 0,C 180,E1 -1370.305,E2 -1370.305} C_VEL
LIN {X 0,Y 587.327,Z 417.948,A -85,B 0,C 180,E1 -1373.259,E2 -1373.259} C_VEL
LIN {X 0,Y 587.34,Z 417.95,A -85,B 0,C 180,E1 -1375.516,E2 -1375.516} C_VEL
LIN {X 0,Y 587.352,Z 417.948,A -85,B 0,C 180,E1 -1377.818,E2 -1377.818} C_VEL
LIN {X 0,Y 587.346,Z 417.942,A -85,B 0,C 180,E1 -1380.511,E2 -1380.511} C_VEL
LIN {X 0,Y 587.343,Z 417.943,A -85,B 0,C 180,E1 -1383.112,E2 -1383.112} C_VEL
LIN {X 0,Y 587.35,Z 417.947,A -85,B 0,C 180,E1 -1385.896,E2 -1385.896} C_VEL
LIN {X 0,Y 587.336,Z 417.942,A -85,B 0,C 180,E1 -1388.479,E2 -1388.479} C_VEL
LIN {X 0,Y 587.34,Z 417.945,A -85,B 0,C 180,E1 -1391.157,E2 -1391.157} C_VEL
LIN {X 0,Y 587.337,Z 417.946,A -85,B 0,C 180,E1 -1394.114,E2 -1394.114} C_VEL
LIN {X 0,Y 587.317,Z 417.946,A -85,B 0,C 180,E1 -1396.993,E2 -1396.993} C_VEL
LIN {X 0,Y 587.322,Z 417.954,A -85,B 0,C 180,E1 -1399.746,E2 -1399.746} C_VEL
LIN {X 0,Y 587.346,Z 417.942,A -85,B 0,C 180,E1 -1402.392,E2 -1402.392} C_VEL
LIN {X 0,Y 587.351,Z 417.941,A -85,B 0,C 180,E1 -1404.946,E2 -1404.946} C_VEL
LIN {X 0,Y 587.341,Z 417.948,A -85,B 0,C 180,E1 -1407.421,E2 -1407.421} C_VEL
LIN {X 0,Y 587.335,Z 417.95,A -85,B 0,C 180,E1 -1409.83,E2 -1409.83} C_VEL
LIN {X 0,Y 587.353,Z 417.942,A -85,B 0,C 180,E1 -1412.307,E2 -1412.307} C_VEL
LIN {X 0,Y 587.339,Z 417.942,A -85,B 0,C 180,E1 -1414.483,E2 -1414.483} C_VEL
LIN {X 0,Y 587.341,Z 417.948,A -85,B 0,C 180,E1 -1417.486,E2 -1417.486} C_VEL
LIN {X 0,Y 587.344,Z 417.942,A -85,B 0,C 180,E1 -1420.425,E2 -1420.425} C_VEL
LIN {X 0,Y 587.355,Z 417.944,A -85,B 0,C 180,E1 -1423.311,E2 -1423.311} C_VEL
LIN {X 0,Y 587.358,Z 417.943,A -85,B 0,C 180,E1 -1426.154,E2 -1426.154} C_VEL
LIN {X 0,Y 587.342,Z 417.942,A -85,B 0,C 180,E1 -1428.962,E2 -1428.962} C_VEL
LIN {X 0,Y 587.371,Z 417.948,A -85,B 0,C 180,E1 -1431.745,E2 -1431.745} C_VEL
LIN {X 0,Y 587.355,Z 417.94,A -85,B 0,C 180,E1 -1434.507,E2 -1434.507} C_VEL
LIN {X 0,Y 587.377,Z 417.94,A -85,B 0,C 180,E1 -1437.257,E2 -1437.257} C_VEL
LIN {X 0,Y 587.382,Z 417.942,A -85,B 0,C 180,E1 -1440,E2 -1440} C_VEL
LIN {X 0,Y 587.377,Z 417.937,A -85,B 0,C 180,E1 -1442.743,E2 -1442.743} C_VEL
LIN {X 0,Y 587.353,Z 417.945,A -85,B 0,C 180,E1 -1445.493,E2 -1445.493} C_VEL
LIN {X 0,Y 587.371,Z 417.94,A -85,B 0,C 180,E1 -1448.255,E2 -1448.255} C_VEL
LIN {X 0,Y 587.347,Z 417.943,A -85,B 0,C 180,E1 -1451.134,E2 -1451.134} C_VEL
LIN {X 0,Y 587.364,Z 417.941,A -85,B 0,C 180,E1 -1454.26,E2 -1454.26} C_VEL
LIN {X 0,Y 587.349,Z 417.946,A -85,B 0,C 180,E1 -1457.406,E2 -1457.406} C_VEL
LIN {X 0,Y 587.329,Z 417.945,A -85,B 0,C 180,E1 -1460.305,E2 -1460.305} C_VEL
LIN {X 0,Y 587.321,Z 417.948,A -85,B 0,C 180,E1 -1463.259,E2 -1463.259} C_VEL
LIN {X 0,Y 587.337,Z 417.95,A -85,B 0,C 180,E1 -1465.516,E2 -1465.516} C_VEL
LIN {X 0,Y 587.348,Z 417.95,A -85,B 0,C 180,E1 -1467.818,E2 -1467.818} C_VEL
LIN {X 0,Y 587.335,Z 417.943,A -85,B 0,C 180,E1 -1470.51,E2 -1470.51} C_VEL
LIN {X 0,Y 587.334,Z 417.948,A -85,B 0,C 180,E1 -1473.397,E2 -1473.397} C_VEL
LIN {X 0,Y 587.356,Z 417.948,A -85,B 0,C 180,E1 -1475.895,E2 -1475.895} C_VEL
LIN {X 0,Y 587.33,Z 417.944,A -85,B 0,C 180,E1 -1478.479,E2 -1478.479} C_VEL
LIN {X 0,Y 587.334,Z 417.945,A -85,B 0,C 180,E1 -1481.157,E2 -1481.157} C_VEL
LIN {X 0,Y 587.326,Z 417.948,A -85,B 0,C 180,E1 -1484.113,E2 -1484.113} C_VEL
LIN {X 0,Y 587.323,Z 417.945,A -85,B 0,C 180,E1 -1486.994,E2 -1486.994} C_VEL
LIN {X 0,Y 587.314,Z 417.956,A -85,B 0,C 180,E1 -1489.746,E2 -1489.746} C_VEL
LIN {X 0,Y 587.346,Z 417.943,A -85,B 0,C 180,E1 -1492.392,E2 -1492.392} C_VEL
LIN {X 0,Y 587.361,Z 417.95,A -85,B 0,C 180,E1 -1495.78,E2 -1495.78} C_VEL
LIN {X 0,Y 587.348,Z 417.945,A -85,B 0,C 180,E1 -1498.231,E2 -1498.231} C_VEL
LIN {X 0,Y 587.349,Z 417.943,A -85,B 0,C 180,E1 -1500.867,E2 -1500.867} C_VEL
LIN {X 0,Y 587.359,Z 417.95,A -85,B 0,C 180,E1 -1503.819,E2 -1503.819} C_VEL
LIN {X 0,Y 587.389,Z 418.178,A -85,B 0,C 180,E1 -1504.105,E2 -1504.105} C_VEL
LIN {X 0,Y 588.289,Z 423.016,A -85,B 0,C 180,E1 -1504.736,E2 -1504.736} C_VEL
LIN {X 0,Y 588.055,Z 446.269,A -85,B 0,C 180,E1 -1507.515,E2 -1507.515} C_VEL
LIN {X 0,Y 587.843,Z 471.239,A -85,B 0,C 180,E1 -1510.442,E2 -1510.442} C_VEL
LIN {X 0,Y 587.811,Z 475.138,A -85,B 0,C 180,E1 -1510.872,E2 -1510.872} C_VEL
LIN {X 0,Y 588.596,Z 479.512,A -85,B 0,C 180,E1 -1510.954,E2 -1510.954} C_VEL
LIN {X 0,Y 588.303,Z 641.318,A -85,B 0,C 180,E1 -1512.998,E2 -1512.998} C_VEL
LIN {X 0,Y 588.211,Z 656.702,A -85,B 0,C 180,E1 -1513.336,E2 -1513.336} C_VEL
LIN {X 0,Y 588.069,Z 672.04,A -85,B 0,C 180,E1 -1513.823,E2 -1513.823} C_VEL
LIN {X 0,Y 587.987,Z 685.759,A -85,B 0,C 180,E1 -1514.399,E2 -1514.399} C_VEL
LIN {X 0,Y 587.829,Z 699.234,A -85,B 0,C 180,E1 -1515.105,E2 -1515.105} C_VEL
LIN {X 0,Y 587.741,Z 712.11,A -85,B 0,C 180,E1 -1515.929,E2 -1515.929} C_VEL
LIN {X 0,Y 587.582,Z 724.284,A -85,B 0,C 180,E1 -1516.864,E2 -1516.864} C_VEL
LIN {X 0,Y 587.454,Z 735.746,A -85,B 0,C 180,E1 -1517.915,E2 -1517.915} C_VEL
LIN {X 0,Y 587.348,Z 745.388,A -85,B 0,C 180,E1 -1518.962,E2 -1518.962} C_VEL
LIN {X 0,Y 587.305,Z 754.854,A -85,B 0,C 180,E1 -1520.182,E2 -1520.182} C_VEL
LIN {X 0,Y 587.264,Z 762.73,A -85,B 0,C 180,E1 -1521.396,E2 -1521.396} C_VEL
LIN {X 0,Y 587.216,Z 770.087,A -85,B 0,C 180,E1 -1522.78,E2 -1522.78} C_VEL
LIN {X 0,Y 587.224,Z 775.923,A -85,B 0,C 180,E1 -1524.161,E2 -1524.161} C_VEL
LIN {X 0,Y 587.136,Z 779.383,A -85,B 0,C 180,E1 -1525.193,E2 -1525.193} C_VEL
LIN {X 0,Y 587.179,Z 782.887,A -85,B 0,C 180,E1 -1526.569,E2 -1526.569} C_VEL
LIN {X 0,Y 587.137,Z 785.193,A -85,B 0,C 180,E1 -1527.942,E2 -1527.942} C_VEL
LIN {X 0,Y 587.137,Z 786.35,A -85,B 0,C 180,E1 -1529.314,E2 -1529.314} C_VEL
LIN {X 0,Y 587.137,Z 786.35,A -85,B 0,C 180,E1 -1530.685,E2 -1530.685} C_VEL
LIN {X 0,Y 587.137,Z 785.193,A -85,B 0,C 180,E1 -1532.058,E2 -1532.058} C_VEL
LIN {X 0,Y 587.179,Z 782.887,A -85,B 0,C 180,E1 -1533.431,E2 -1533.431} C_VEL
LIN {X 0,Y 587.136,Z 779.385,A -85,B 0,C 180,E1 -1534.806,E2 -1534.806} C_VEL
LIN {X 0,Y 587.178,Z 774.61,A -85,B 0,C 180,E1 -1536.184,E2 -1536.184} C_VEL
LIN {X 0,Y 587.235,Z 768.427,A -85,B 0,C 180,E1 -1537.564,E2 -1537.564} C_VEL
LIN {X 0,Y 587.266,Z 760.654,A -85,B 0,C 180,E1 -1538.95,E2 -1538.95} C_VEL
LIN {X 0,Y 587.351,Z 752.373,A -85,B 0,C 180,E1 -1540.165,E2 -1540.165} C_VEL
LIN {X 0,Y 587.399,Z 742.399,A -85,B 0,C 180,E1 -1541.385,E2 -1541.385} C_VEL
LIN {X 0,Y 587.521,Z 732.196,A -85,B 0,C 180,E1 -1542.434,E2 -1542.434} C_VEL
LIN {X 0,Y 587.629,Z 720.024,A -85,B 0,C 180,E1 -1543.486,E2 -1543.486} C_VEL
LIN {X 0,Y 587.773,Z 707.064,A -85,B 0,C 180,E1 -1544.416,E2 -1544.416} C_VEL
LIN {X 0,Y 587.886,Z 692.876,A -85,B 0,C 180,E1 -1545.248,E2 -1545.248} C_VEL
LIN {X 0,Y 588.049,Z 678.81,A -85,B 0,C 180,E1 -1545.91,E2 -1545.91} C_VEL
LIN {X 0,Y 588.168,Z 664.321,A -85,B 0,C 180,E1 -1546.441,E2 -1546.441} C_VEL
LIN {X 0,Y 588.278,Z 649.297,A -85,B 0,C 180,E1 -1546.844,E2 -1546.844} C_VEL
LIN {X 0,Y 588.32,Z 634.107,A -85,B 0,C 180,E1 -1547.11,E2 -1547.11} C_VEL
LIN {X 0,Y 588.501,Z 478.542,A -85,B 0,C 180,E1 -1549.062,E2 -1549.062} C_VEL
LIN {X 0,Y 587.805,Z 474.774,A -85,B 0,C 180,E1 -1549.148,E2 -1549.148} C_VEL
LIN {X 0,Y 588.008,Z 450.958,A -85,B 0,C 180,E1 -1551.931,E2 -1551.931} C_VEL
LIN {X 0,Y 588.258,Z 427.092,A -85,B 0,C 180,E1 -1554.772,E2 -1554.772} C_VEL
LIN {X 0,Y 588.117,Z 421.306,A -85,B 0,C 180,E1 -1555.48,E2 -1555.48} C_VEL
LIN {X 0,Y 587.338,Z 417.952,A -85,B 0,C 180,E1 -1555.949,E2 -1555.949} C_VEL
LIN {X 0,Y 587.325,Z 417.951,A -85,B 0,C 180,E1 -1558.596,E2 -1558.596} C_VEL
LIN {X 0,Y 587.339,Z 417.944,A -85,B 0,C 180,E1 -1560.965,E2 -1560.965} C_VEL
LIN {X 0,Y 587.332,Z 417.944,A -85,B 0,C 180,E1 -1563.396,E2 -1563.396} C_VEL
LIN {X 0,Y 587.315,Z 417.95,A -85,B 0,C 180,E1 -1565.897,E2 -1565.897} C_VEL
LIN {X 0,Y 587.33,Z 417.951,A -85,B 0,C 180,E1 -1568.478,E2 -1568.478} C_VEL
LIN {X 0,Y 587.333,Z 417.944,A -85,B 0,C 180,E1 -1571.156,E2 -1571.156} C_VEL
LIN {X 0,Y 587.329,Z 417.951,A -85,B 0,C 180,E1 -1574.114,E2 -1574.114} C_VEL
LIN {X 0,Y 587.309,Z 417.947,A -85,B 0,C 180,E1 -1576.993,E2 -1576.993} C_VEL
LIN {X 0,Y 587.314,Z 417.948,A -85,B 0,C 180,E1 -1579.746,E2 -1579.746} C_VEL
LIN {X 0,Y 587.338,Z 417.952,A -85,B 0,C 180,E1 -1582.392,E2 -1582.392} C_VEL
LIN {X 0,Y 587.347,Z 417.943,A -85,B 0,C 180,E1 -1584.946,E2 -1584.946} C_VEL
LIN {X 0,Y 587.334,Z 417.943,A -85,B 0,C 180,E1 -1587.421,E2 -1587.421} C_VEL
LIN {X 0,Y 587.328,Z 417.946,A -85,B 0,C 180,E1 -1589.83,E2 -1589.83} C_VEL
LIN {X 0,Y 587.344,Z 417.952,A -85,B 0,C 180,E1 -1592.306,E2 -1592.306} C_VEL
LIN {X 0,Y 587.335,Z 417.951,A -85,B 0,C 180,E1 -1594.484,E2 -1594.484} C_VEL
LIN {X 0,Y 587.333,Z 417.943,A -85,B 0,C 180,E1 -1597.486,E2 -1597.486} C_VEL
LIN {X 0,Y 587.326,Z 417.945,A -85,B 0,C 180,E1 -1599.695,E2 -1599.695} C_VEL
LIN {X 0,Y 587.351,Z 417.947,A -85,B 0,C 180,E1 -1602.594,E2 -1602.594} C_VEL
LIN {X 0,Y 587.357,Z 417.942,A -85,B 0,C 180,E1 -1605.739,E2 -1605.739} C_VEL
LIN {X 0,Y 587.336,Z 417.951,A -85,B 0,C 180,E1 -1608.263,E2 -1608.263} C_VEL
LIN {X 0,Y 587.34,Z 417.943,A -85,B 0,C 180,E1 -1611.051,E2 -1611.051} C_VEL
LIN {X 0,Y 587.368,Z 417.939,A -85,B 0,C 180,E1 -1613.264,E2 -1613.264} C_VEL
LIN {X 0,Y 587.316,Z 417.948,A -85,B 0,C 180,E1 -1615.883,E2 -1615.883} C_VEL
LIN {X 0,Y 587.363,Z 417.943,A -85,B 0,C 180,E1 -1617.943,E2 -1617.943} C_VEL
LIN {X 0,Y 587.389,Z 417.941,A -85,B 0,C 180,E1 -1620.686,E2 -1620.686} C_VEL
LIN {X 0,Y 587.33,Z 417.944,A -85,B 0,C 180,E1 -1623.43,E2 -1623.43} C_VEL
LIN {X 0,Y 587.356,Z 417.94,A -85,B 0,C 180,E1 -1625.493,E2 -1625.493} C_VEL
LIN {X 0,Y 587.367,Z 417.947,A -85,B 0,C 180,E1 -1628.255,E2 -1628.255} C_VEL
LIN {X 0,Y 587.34,Z 417.943,A -85,B 0,C 180,E1 -1631.134,E2 -1631.134} C_VEL
LIN {X 0,Y 587.353,Z 417.943,A -85,B 0,C 180,E1 -1633.846,E2 -1633.846} C_VEL
LIN {X 0,Y 587.359,Z 417.944,A -85,B 0,C 180,E1 -1636.82,E2 -1636.82} C_VEL
LIN {X 0,Y 587.322,Z 417.948,A -85,B 0,C 180,E1 -1638.324,E2 -1638.324} C_VEL
LIN {X 0,Y 586.669,Z 418.029,A -85,B 0,C 180,E1 -1638.896,E2 -1638.896} C_VEL
LIN {X 0,Y 583.838,Z 418.38,A -85,B 0,C 180,E1 -1639.824,E2 -1639.824} C_VEL
LIN {X 0,Y 581.428,Z 418.687,A -85,B 0,C 180,E1 -1640.571,E2 -1640.571} C_VEL
LIN {X 0,Y 580.376,Z 418.811,A -85,B 0,C 180,E1 -1641.148,E2 -1641.148} C_VEL
LIN {X 0,Y 580.282,Z 418.822,A -85,B 0,C 180,E1 -1641.343,E2 -1641.343} C_VEL
LIN {X 0,Y 580.276,Z 418.823,A -85,B 0,C 180,E1 -1643.558,E2 -1643.558} C_VEL
LIN {X 0,Y 580.324,Z 418.826,A -85,B 0,C 180,E1 -1646.343,E2 -1646.343} C_VEL
LIN {X 0,Y 580.304,Z 418.819,A -85,B 0,C 180,E1 -1649.312,E2 -1649.312} C_VEL
LIN {X 0,Y 580.301,Z 418.826,A -85,B 0,C 180,E1 -1652.201,E2 -1652.201} C_VEL
LIN {X 0,Y 580.298,Z 418.826,A -85,B 0,C 180,E1 -1654.696,E2 -1654.696} C_VEL
LIN {X 0,Y 580.296,Z 418.821,A -85,B 0,C 180,E1 -1657.269,E2 -1657.269} C_VEL
LIN {X 0,Y 580.303,Z 418.828,A -85,B 0,C 180,E1 -1660.273,E2 -1660.273} C_VEL
LIN {X 0,Y 580.274,Z 418.831,A -85,B 0,C 180,E1 -1662.707,E2 -1662.707} C_VEL
LIN {X 0,Y 580.339,Z 418.96,A -85,B 0,C 180,E1 -1664.95,E2 -1664.95} C_VEL
LIN {X 0,Y 581.024,Z 422.943,A -85,B 0,C 180,E1 -1665.534,E2 -1665.534} C_VEL
LIN {X 0,Y 580.781,Z 444.452,A -85,B 0,C 180,E1 -1668.483,E2 -1668.483} C_VEL
LIN {X 0,Y 580.771,Z 446.051,A -85,B 0,C 180,E1 -1668.688,E2 -1668.688} C_VEL
LIN {X 0,Y 581.89,Z 452.284,A -85,B 0,C 180,E1 -1668.806,E2 -1668.806} C_VEL
LIN {X 0,Y 581.526,Z 611.349,A -85,B 0,C 180,E1 -1670.84,E2 -1670.84} C_VEL
LIN {X 0,Y 581.399,Z 627.08,A -85,B 0,C 180,E1 -1671.191,E2 -1671.191} C_VEL
LIN {X 0,Y 581.269,Z 641.07,A -85,B 0,C 180,E1 -1671.638,E2 -1671.638} C_VEL
LIN {X 0,Y 581.118,Z 655.617,A -85,B 0,C 180,E1 -1672.248,E2 -1672.248} C_VEL
LIN {X 0,Y 580.916,Z 669.533,A -85,B 0,C 180,E1 -1672.985,E2 -1672.985} C_VEL
LIN {X 0,Y 580.786,Z 683.109,A -85,B 0,C 180,E1 -1673.872,E2 -1673.872} C_VEL
LIN {X 0,Y 580.592,Z 696.117,A -85,B 0,C 180,E1 -1674.903,E2 -1674.903} C_VEL
LIN {X 0,Y 580.459,Z 707.093,A -85,B 0,C 180,E1 -1675.947,E2 -1675.947} C_VEL
LIN {X 0,Y 580.335,Z 717.992,A -85,B 0,C 180,E1 -1677.186,E2 -1677.186} C_VEL
LIN {X 0,Y 580.25,Z 726.978,A -85,B 0,C 180,E1 -1678.41,E2 -1678.41} C_VEL
LIN {X 0,Y 580.17,Z 735.49,A -85,B 0,C 180,E1 -1679.821,E2 -1679.821} C_VEL
LIN {X 0,Y 580.111,Z 741.371,A -85,B 0,C 180,E1 -1681.015,E2 -1681.015} C_VEL
LIN {X 0,Y 580.077,Z 746.101,A -85,B 0,C 180,E1 -1682.183,E2 -1682.183} C_VEL
LIN {X 0,Y 580.097,Z 750.854,A -85,B 0,C 180,E1 -1683.706,E2 -1683.706} C_VEL
LIN {X 0,Y 580.043,Z 754.287,A -85,B 0,C 180,E1 -1685.331,E2 -1685.331} C_VEL
LIN {X 0,Y 580.025,Z 755.721,A -85,B 0,C 180,E1 -1686.432,E2 -1686.432} C_VEL
LIN {X 0,Y 580.032,Z 756.482,A -85,B 0,C 180,E1 -1687.938,E2 -1687.938} C_VEL
LIN {X 0,Y 580.045,Z 755.915,A -85,B 0,C 180,E1 -1689.429,E2 -1689.429} C_VEL
LIN {X 0,Y 580.067,Z 754.038,A -85,B 0,C 180,E1 -1690.916,E2 -1690.916} C_VEL
LIN {X 0,Y 580.045,Z 750.897,A -85,B 0,C 180,E1 -1692.368,E2 -1692.368} C_VEL
LIN {X 0,Y 580.109,Z 746.401,A -85,B 0,C 180,E1 -1693.821,E2 -1693.821} C_VEL
LIN {X 0,Y 580.147,Z 740.505,A -85,B 0,C 180,E1 -1695.263,E2 -1695.263} C_VEL
LIN {X 0,Y 580.203,Z 733.072,A -85,B 0,C 180,E1 -1696.695,E2 -1696.695} C_VEL
LIN {X 0,Y 580.289,Z 725.149,A -85,B 0,C 180,E1 -1697.942,E2 -1697.942} C_VEL
LIN {X 0,Y 580.36,Z 715.53,A -85,B 0,C 180,E1 -1699.2,E2 -1699.2} C_VEL
LIN {X 0,Y 580.492,Z 704.34,A -85,B 0,C 180,E1 -1700.418,E2 -1700.418} C_VEL
LIN {X 0,Y 580.628,Z 692.71,A -85,B 0,C 180,E1 -1701.473,E2 -1701.473} C_VEL
LIN {X 0,Y 580.792,Z 679.952,A -85,B 0,C 180,E1 -1702.439,E2 -1702.439} C_VEL
LIN {X 0,Y 580.993,Z 666.566,A -85,B 0,C 180,E1 -1703.273,E2 -1703.273} C_VEL
LIN {X 0,Y 581.143,Z 653.759,A -85,B 0,C 180,E1 -1703.926,E2 -1703.926} C_VEL
LIN {X 0,Y 581.297,Z 639.861,A -85,B 0,C 180,E1 -1704.494,E2 -1704.494} C_VEL
LIN {X 0,Y 581.446,Z 625.012,A -85,B 0,C 180,E1 -1704.951,E2 -1704.951} C_VEL
LIN {X 0,Y 581.506,Z 611.065,A -85,B 0,C 180,E1 -1705.256,E2 -1705.256} C_VEL
LIN {X 0,Y 581.777,Z 450.821,A -85,B 0,C 180,E1 -1707.307,E2 -1707.307} C_VEL
LIN {X 0,Y 580.764,Z 445.818,A -85,B 0,C 180,E1 -1707.421,E2 -1707.421} C_VEL
LIN {X 0,Y 580.971,Z 425.716,A -85,B 0,C 180,E1 -1710.174,E2 -1710.174} C_VEL
LIN {X 0,Y 580.725,Z 420.798,A -85,B 0,C 180,E1 -1710.867,E2 -1710.867} C_VEL
LIN {X 0,Y 580.345,Z 418.823,A -85,B 0,C 180,E1 -1711.171,E2 -1711.171} C_VEL
LIN {X 0,Y 580.291,Z 418.83,A -85,B 0,C 180,E1 -1713.472,E2 -1713.472} C_VEL
LIN {X 0,Y 580.327,Z 418.825,A -85,B 0,C 180,E1 -1715.56,E2 -1715.56} C_VEL
LIN {X 0,Y 580.332,Z 418.817,A -85,B 0,C 180,E1 -1718.356,E2 -1718.356} C_VEL
LIN {X 0,Y 580.305,Z 418.821,A -85,B 0,C 180,E1 -1721.191,E2 -1721.191} C_VEL
LIN {X 0,Y 580.332,Z 418.82,A -85,B 0,C 180,E1 -1724.017,E2 -1724.017} C_VEL
LIN {X 0,Y 580.317,Z 418.818,A -85,B 0,C 180,E1 -1726.914,E2 -1726.914} C_VEL
LIN {X 0,Y 580.309,Z 418.826,A -85,B 0,C 180,E1 -1729.822,E2 -1729.822} C_VEL
LIN {X 0,Y 580.299,Z 418.82,A -85,B 0,C 180,E1 -1732.802,E2 -1732.802} C_VEL
LIN {X 0,Y 580.312,Z 418.819,A -85,B 0,C 180,E1 -1735.08,E2 -1735.08} C_VEL
LIN {X 0,Y 580.304,Z 418.82,A -85,B 0,C 180,E1 -1738.185,E2 -1738.185} C_VEL
LIN {X 0,Y 580.297,Z 418.82,A -85,B 0,C 180,E1 -1740.696,E2 -1740.696} C_VEL
LIN {X 0,Y 580.308,Z 418.822,A -85,B 0,C 180,E1 -1743.316,E2 -1743.316} C_VEL
LIN {X 0,Y 580.296,Z 418.82,A -85,B 0,C 180,E1 -1746.402,E2 -1746.402} C_VEL
LIN {X 0,Y 580.31,Z 418.82,A -85,B 0,C 180,E1 -1749.187,E2 -1749.187} C_VEL
LIN {X 0,Y 580.317,Z 418.825,A -85,B 0,C 180,E1 -1751.765,E2 -1751.765} C_VEL
LIN {X 0,Y 580.271,Z 418.823,A -85,B 0,C 180,E1 -1754.625,E2 -1754.625} C_VEL
LIN {X 0,Y 580.288,Z 418.831,A -85,B 0,C 180,E1 -1757.628,E2 -1757.628} C_VEL
LIN {X 0,Y 580.297,Z 418.823,A -85,B 0,C 180,E1 -1760.067,E2 -1760.067} C_VEL
LIN {X 0,Y 580.303,Z 418.82,A -85,B 0,C 180,E1 -1763.065,E2 -1763.065} C_VEL
LIN {X 0,Y 580.305,Z 418.824,A -85,B 0,C 180,E1 -1765.44,E2 -1765.44} C_VEL
LIN {X 0,Y 580.305,Z 418.824,A -85,B 0,C 180,E1 -1767.969,E2 -1767.969} C_VEL
LIN {X 0,Y 580.304,Z 418.817,A -85,B 0,C 180,E1 -1770.69,E2 -1770.69} C_VEL
LIN {X 0,Y 580.329,Z 418.826,A -85,B 0,C 180,E1 -1773.658,E2 -1773.658} C_VEL
LIN {X 0,Y 580.28,Z 418.82,A -85,B 0,C 180,E1 -1776.442,E2 -1776.442} C_VEL
LIN {X 0,Y 580.277,Z 418.828,A -85,B 0,C 180,E1 -1779.437,E2 -1779.437} C_VEL
LIN {X 0,Y 580.27,Z 418.833,A -85,B 0,C 180,E1 -1781.645,E2 -1781.645} C_VEL
LIN {X 0,Y 580.282,Z 418.829,A -85,B 0,C 180,E1 -1783.825,E2 -1783.825} C_VEL
LIN {X 0,Y 580.325,Z 418.821,A -85,B 0,C 180,E1 -1785.983,E2 -1785.983} C_VEL
LIN {X 0,Y 580.304,Z 418.818,A -85,B 0,C 180,E1 -1788.827,E2 -1788.827} C_VEL
LIN {X 0,Y 580.335,Z 418.823,A -85,B 0,C 180,E1 -1791.644,E2 -1791.644} C_VEL
LIN {X 0,Y 580.322,Z 418.817,A -85,B 0,C 180,E1 -1794.44,E2 -1794.44} C_VEL
LIN {X 0,Y 580.343,Z 418.815,A -85,B 0,C 180,E1 -1797.223,E2 -1797.223} C_VEL
LIN {X 0,Y 580.352,Z 418.818,A -85,B 0,C 180,E1 -1800,E2 -1800} C_VEL
LIN {X 0,Y 580.343,Z 418.813,A -85,B 0,C 180,E1 -1802.776,E2 -1802.776} C_VEL
LIN {X 0,Y 580.32,Z 418.822,A -85,B 0,C 180,E1 -1805.56,E2 -1805.56} C_VEL
LIN {X 0,Y 580.334,Z 418.816,A -85,B 0,C 180,E1 -1808.356,E2 -1808.356} C_VEL
LIN {X 0,Y 580.299,Z 418.821,A -85,B 0,C 180,E1 -1811.191,E2 -1811.191} C_VEL
LIN {X 0,Y 580.324,Z 418.821,A -85,B 0,C 180,E1 -1814.017,E2 -1814.017} C_VEL
LIN {X 0,Y 580.311,Z 418.818,A -85,B 0,C 180,E1 -1816.914,E2 -1816.914} C_VEL
LIN {X 0,Y 580.304,Z 418.827,A -85,B 0,C 180,E1 -1819.822,E2 -1819.822} C_VEL
LIN {X 0,Y 580.294,Z 418.82,A -85,B 0,C 180,E1 -1822.802,E2 -1822.802} C_VEL
LIN {X 0,Y 580.307,Z 418.82,A -85,B 0,C 180,E1 -1825.08,E2 -1825.08} C_VEL
LIN {X 0,Y 580.301,Z 418.822,A -85,B 0,C 180,E1 -1828.185,E2 -1828.185} C_VEL
LIN {X 0,Y 580.282,Z 418.821,A -85,B 0,C 180,E1 -1830.694,E2 -1830.694} C_VEL
LIN {X 0,Y 580.303,Z 418.823,A -85,B 0,C 180,E1 -1833.316,E2 -1833.316} C_VEL
LIN {X 0,Y 580.326,Z 418.826,A -85,B 0,C 180,E1 -1835.767,E2 -1835.767} C_VEL
LIN {X 0,Y 580.287,Z 418.824,A -85,B 0,C 180,E1 -1838.146,E2 -1838.146} C_VEL
LIN {X 0,Y 580.298,Z 418.82,A -85,B 0,C 180,E1 -1840.843,E2 -1840.843} C_VEL
LIN {X 0,Y 580.278,Z 418.832,A -85,B 0,C 180,E1 -1843.658,E2 -1843.658} C_VEL
LIN {X 0,Y 580.286,Z 418.821,A -85,B 0,C 180,E1 -1846.608,E2 -1846.608} C_VEL
LIN {X 0,Y 580.299,Z 418.822,A -85,B 0,C 180,E1 -1849.157,E2 -1849.157} C_VEL
LIN {X 0,Y 580.291,Z 418.828,A -85,B 0,C 180,E1 -1851.927,E2 -1851.927} C_VEL
LIN {X 0,Y 580.251,Z 418.827,A -85,B 0,C 180,E1 -1854.453,E2 -1854.453} C_VEL
LIN {X 0,Y 580.291,Z 418.822,A -85,B 0,C 180,E1 -1856.975,E2 -1856.975} C_VEL
LIN {X 0,Y 580.3,Z 418.826,A -85,B 0,C 180,E1 -1859.425,E2 -1859.425} C_VEL
LIN {X 0,Y 580.298,Z 418.827,A -85,B 0,C 180,E1 -1862.141,E2 -1862.141} C_VEL
LIN {X 0,Y 580.332,Z 418.881,A -85,B 0,C 180,E1 -1863.854,E2 -1863.854} C_VEL
LIN {X 0,Y 581.469,Z 424.42,A -85,B 0,C 180,E1 -1864.591,E2 -1864.591} C_VEL
LIN {X 0,Y 581.208,Z 447.83,A -85,B 0,C 180,E1 -1867.423,E2 -1867.423} C_VEL
LIN {X 0,Y 580.922,Z 472.547,A -85,B 0,C 180,E1 -1870.354,E2 -1870.354} C_VEL
LIN {X 0,Y 580.898,Z 474.902,A -85,B 0,C 180,E1 -1870.63,E2 -1870.63} C_VEL
LIN {X 0,Y 581.876,Z 480.694,A -85,B 0,C 180,E1 -1870.74,E2 -1870.74} C_VEL
LIN {X 0,Y 581.531,Z 641.445,A -85,B 0,C 180,E1 -1872.797,E2 -1872.797} C_VEL
LIN {X 0,Y 581.415,Z 656.701,A -85,B 0,C 180,E1 -1873.135,E2 -1873.135} C_VEL
LIN {X 0,Y 581.244,Z 672.038,A -85,B 0,C 180,E1 -1873.627,E2 -1873.627} C_VEL
LIN {X 0,Y 581.123,Z 685.762,A -85,B 0,C 180,E1 -1874.21,E2 -1874.21} C_VEL
LIN {X 0,Y 580.944,Z 699.236,A -85,B 0,C 180,E1 -1874.924,E2 -1874.924} C_VEL
LIN {X 0,Y 580.805,Z 712.475,A -85,B 0,C 180,E1 -1875.783,E2 -1875.783} C_VEL
LIN {X 0,Y 580.608,Z 724.285,A -85,B 0,C 180,E1 -1876.704,E2 -1876.704} C_VEL
LIN {X 0,Y 580.479,Z 735.746,A -85,B 0,C 180,E1 -1877.767,E2 -1877.767} C_VEL
LIN {X 0,Y 580.308,Z 746.453,A -85,B 0,C 180,E1 -1878.953,E2 -1878.953} C_VEL
LIN {X 0,Y 580.268,Z 754.855,A -85,B 0,C 180,E1 -1880.061,E2 -1880.061} C_VEL
LIN {X 0,Y 580.214,Z 762.731,A -85,B 0,C 180,E1 -1881.291,E2 -1881.291} C_VEL
LIN {X 0,Y 580.131,Z 770.087,A -85,B 0,C 180,E1 -1882.692,E2 -1882.692} C_VEL
LIN {X 0,Y 580.129,Z 775.923,A -85,B 0,C 180,E1 -1884.089,E2 -1884.089} C_VEL
LIN {X 0,Y 580.041,Z 779.383,A -85,B 0,C 180,E1 -1885.134,E2 -1885.134} C_VEL
LIN {X 0,Y 580.105,Z 782.887,A -85,B 0,C 180,E1 -1886.527,E2 -1886.527} C_VEL
LIN {X 0,Y 580.036,Z 785.193,A -85,B 0,C 180,E1 -1887.917,E2 -1887.917} C_VEL
LIN {X 0,Y 580.038,Z 786.349,A -85,B 0,C 180,E1 -1889.305,E2 -1889.305} C_VEL
LIN {X 0,Y 580.038,Z 786.349,A -85,B 0,C 180,E1 -1890.694,E2 -1890.694} C_VEL
LIN {X 0,Y 580.036,Z 785.192,A -85,B 0,C 180,E1 -1892.083,E2 -1892.083} C_VEL
LIN {X 0,Y 580.105,Z 782.887,A -85,B 0,C 180,E1 -1893.472,E2 -1893.472} C_VEL
LIN {X 0,Y 580.041,Z 779.386,A -85,B 0,C 180,E1 -1894.865,E2 -1894.865} C_VEL
LIN {X 0,Y 580.091,Z 774.61,A -85,B 0,C 180,E1 -1896.259,E2 -1896.259} C_VEL
LIN {X 0,Y 580.168,Z 768.426,A -85,B 0,C 180,E1 -1897.657,E2 -1897.657} C_VEL
LIN {X 0,Y 580.207,Z 760.653,A -85,B 0,C 180,E1 -1899.059,E2 -1899.059} C_VEL
LIN {X 0,Y 580.308,Z 752.373,A -85,B 0,C 180,E1 -1900.29,E2 -1900.29} C_VEL
LIN {X 0,Y 580.382,Z 742.399,A -85,B 0,C 180,E1 -1901.525,E2 -1901.525} C_VEL
LIN {X 0,Y 580.54,Z 732.195,A -85,B 0,C 180,E1 -1902.586,E2 -1902.586} C_VEL
LIN {X 0,Y 580.677,Z 720.025,A -85,B 0,C 180,E1 -1903.651,E2 -1903.651} C_VEL
LIN {X 0,Y 580.844,Z 707.814,A -85,B 0,C 180,E1 -1904.541,E2 -1904.541} C_VEL
LIN {X 0,Y 580.986,Z 694.53,A -85,B 0,C 180,E1 -1905.343,E2 -1905.343} C_VEL
LIN {X 0,Y 581.201,Z 679.848,A -85,B 0,C 180,E1 -1906.057,E2 -1906.057} C_VEL
LIN {X 0,Y 581.34,Z 665.633,A -85,B 0,C 180,E1 -1906.595,E2 -1906.595} C_VEL
LIN {X 0,Y 581.471,Z 651.188,A -85,B 0,C 180,E1 -1907,E2 -1907} C_VEL
LIN {X 0,Y 581.518,Z 636.853,A -85,B 0,C 180,E1 -1907.275,E2 -1907.275} C_VEL
LIN {X 0,Y 581.806,Z 479.516,A -85,B 0,C 180,E1 -1909.277,E2 -1909.277} C_VEL
LIN {X 0,Y 580.919,Z 474.763,A -85,B 0,C 180,E1 -1909.385,E2 -1909.385} C_VEL
LIN {X 0,Y 581.148,Z 450.958,A -85,B 0,C 180,E1 -1912.204,E2 -1912.204} C_VEL
LIN {X 0,Y 581.438,Z 428.03,A -85,B 0,C 180,E1 -1914.968,E2 -1914.968} C_VEL
LIN {X 0,Y 581.26,Z 422.866,A -85,B 0,C 180,E1 -1915.61,E2 -1915.61} C_VEL
LIN {X 0,Y 580.327,Z 418.827,A -85,B 0,C 180,E1 -1916.175,E2 -1916.175} C_VEL
LIN {X 0,Y 580.291,Z 418.824,A -85,B 0,C 180,E1 -1918.975,E2 -1918.975} C_VEL
LIN {X 0,Y 580.286,Z 418.822,A -85,B 0,C 180,E1 -1921.384,E2 -1921.384} C_VEL
LIN {X 0,Y 580.313,Z 418.822,A -85,B 0,C 180,E1 -1923.854,E2 -1923.854} C_VEL
LIN {X 0,Y 580.299,Z 418.821,A -85,B 0,C 180,E1 -1926.934,E2 -1926.934} C_VEL
LIN {X 0,Y 580.291,Z 418.825,A -85,B 0,C 180,E1 -1929.932,E2 -1929.932} C_VEL
LIN {X 0,Y 580.287,Z 418.824,A -85,B 0,C 180,E1 -1932.704,E2 -1932.704} C_VEL
LIN {X 0,Y 580.264,Z 418.825,A -85,B 0,C 180,E1 -1935.608,E2 -1935.608} C_VEL
LIN {X 0,Y 580.308,Z 418.827,A -85,B 0,C 180,E1 -1938.234,E2 -1938.234} C_VEL
LIN {X 0,Y 580.284,Z 418.823,A -85,B 0,C 180,E1 -1940.966,E2 -1940.966} C_VEL
LIN {X 0,Y 580.29,Z 418.822,A -85,B 0,C 180,E1 -1943.598,E2 -1943.598} C_VEL
LIN {X 0,Y 580.314,Z 418.825,A -85,B 0,C 180,E1 -1946.145,E2 -1946.145} C_VEL
LIN {X 0,Y 580.282,Z 418.827,A -85,B 0,C 180,E1 -1948.615,E2 -1948.615} C_VEL
LIN {X 0,Y 580.289,Z 418.822,A -85,B 0,C 180,E1 -1951.024,E2 -1951.024} C_VEL
LIN {X 0,Y 580.322,Z 418.817,A -85,B 0,C 180,E1 -1953.658,E2 -1953.658} C_VEL
LIN {X 0,Y 580.273,Z 418.831,A -85,B 0,C 180,E1 -1956.442,E2 -1956.442} C_VEL
LIN {X 0,Y 580.276,Z 418.822,A -85,B 0,C 180,E1 -1959.437,E2 -1959.437} C_VEL
LIN {X 0,Y 580.275,Z 418.823,A -85,B 0,C 180,E1 -1961.645,E2 -1961.645} C_VEL
LIN {X 0,Y 580.275,Z 418.824,A -85,B 0,C 180,E1 -1963.826,E2 -1963.826} C_VEL
LIN {X 0,Y 580.318,Z 418.821,A -85,B 0,C 180,E1 -1965.983,E2 -1965.983} C_VEL
LIN {X 0,Y 580.296,Z 418.823,A -85,B 0,C 180,E1 -1968.827,E2 -1968.827} C_VEL
LIN {X 0,Y 580.33,Z 418.816,A -85,B 0,C 180,E1 -1971.644,E2 -1971.644} C_VEL
LIN {X 0,Y 580.317,Z 418.827,A -85,B 0,C 180,E1 -1974.44,E2 -1974.44} C_VEL
LIN {X 0,Y 580.34,Z 418.814,A -85,B 0,C 180,E1 -1977.224,E2 -1977.224} C_VEL
LIN {X 0,Y 580.345,Z 418.818,A -85,B 0,C 180,E1 -1980,E2 -1980} C_VEL
LIN {X 0,Y 580.34,Z 418.818,A -85,B 0,C 180,E1 -1982.777,E2 -1982.777} C_VEL
LIN {X 0,Y 580.323,Z 418.816,A -85,B 0,C 180,E1 -1985.56,E2 -1985.56} C_VEL
LIN {X 0,Y 580.33,Z 418.825,A -85,B 0,C 180,E1 -1988.356,E2 -1988.356} C_VEL
LIN {X 0,Y 580.292,Z 418.82,A -85,B 0,C 180,E1 -1991.191,E2 -1991.191} C_VEL
LIN {X 0,Y 580.319,Z 418.821,A -85,B 0,C 180,E1 -1994.017,E2 -1994.017} C_VEL
LIN {X 0,Y 580.309,Z 418.821,A -85,B 0,C 180,E1 -1996.916,E2 -1996.916} C_VEL
LIN {X 0,Y 580.302,Z 418.821,A -85,B 0,C 180,E1 -1999.823,E2 -1999.823} C_VEL
LIN {X 0,Y 580.282,Z 418.822,A -85,B 0,C 180,E1 -2001.343,E2 -2001.343} C_VEL
LIN {X 0,Y 579.585,Z 418.912,A -85,B 0,C 180,E1 -2001.922,E2 -2001.922} C_VEL
LIN {X 0,Y 576.708,Z 419.271,A -85,B 0,C 180,E1 -2002.862,E2 -2002.862} C_VEL
LIN {X 0,Y 574.312,Z 419.568,A -85,B 0,C 180,E1 -2003.618,E2 -2003.618} C_VEL
LIN {X 0,Y 573.313,Z 419.697,A -85,B 0,C 180,E1 -2004.202,E2 -2004.202} C_VEL
LIN {X 0,Y 573.246,Z 419.703,A -85,B 0,C 180,E1 -2004.399,E2 -2004.399} C_VEL
LIN {X 0,Y 573.26,Z 419.699,A -85,B 0,C 180,E1 -2006.976,E2 -2006.976} C_VEL
LIN {X 0,Y 573.25,Z 419.698,A -85,B 0,C 180,E1 -2009.491,E2 -2009.491} C_VEL
LIN {X 0,Y 573.253,Z 419.705,A -85,B 0,C 180,E1 -2012.23,E2 -2012.23} C_VEL
LIN {X 0,Y 573.249,Z 419.703,A -85,B 0,C 180,E1 -2014.775,E2 -2014.775} C_VEL
LIN {X 0,Y 573.25,Z 419.7,A -85,B 0,C 180,E1 -2017.167,E2 -2017.167} C_VEL
LIN {X 0,Y 573.247,Z 419.7,A -85,B 0,C 180,E1 -2019.607,E2 -2019.607} C_VEL
LIN {X 0,Y 573.237,Z 419.709,A -85,B 0,C 180,E1 -2022.642,E2 -2022.642} C_VEL
LIN {X 0,Y 573.272,Z 419.822,A -85,B 0,C 180,E1 -2024.771,E2 -2024.771} C_VEL
LIN {X 0,Y 574.133,Z 424.663,A -85,B 0,C 180,E1 -2025.49,E2 -2025.49} C_VEL
LIN {X 0,Y 573.853,Z 445.83,A -85,B 0,C 180,E1 -2028.428,E2 -2028.428} C_VEL
LIN {X 0,Y 575.19,Z 453.325,A -85,B 0,C 180,E1 -2028.586,E2 -2028.586} C_VEL
LIN {X 0,Y 574.745,Z 611.375,A -85,B 0,C 180,E1 -2030.631,E2 -2030.631} C_VEL
LIN {X 0,Y 574.594,Z 627.108,A -85,B 0,C 180,E1 -2030.986,E2 -2030.986} C_VEL
LIN {X 0,Y 574.452,Z 641.897,A -85,B 0,C 180,E1 -2031.468,E2 -2031.468} C_VEL
LIN {X 0,Y 574.256,Z 656.698,A -85,B 0,C 180,E1 -2032.106,E2 -2032.106} C_VEL
LIN {X 0,Y 574.026,Z 670.257,A -85,B 0,C 180,E1 -2032.842,E2 -2032.842} C_VEL
LIN {X 0,Y 573.83,Z 684.217,A -85,B 0,C 180,E1 -2033.777,E2 -2033.777} C_VEL
LIN {X 0,Y 573.637,Z 696.068,A -85,B 0,C 180,E1 -2034.736,E2 -2034.736} C_VEL
LIN {X 0,Y 573.445,Z 708.028,A -85,B 0,C 180,E1 -2035.897,E2 -2035.897} C_VEL
LIN {X 0,Y 573.293,Z 717.107,A -85,B 0,C 180,E1 -2036.94,E2 -2036.94} C_VEL
LIN {X 0,Y 573.185,Z 726.234,A -85,B 0,C 180,E1 -2038.182,E2 -2038.182} C_VEL
LIN {X 0,Y 573.118,Z 734.144,A -85,B 0,C 180,E1 -2039.477,E2 -2039.477} C_VEL
LIN {X 0,Y 573.052,Z 739.982,A -85,B 0,C 180,E1 -2040.623,E2 -2040.623} C_VEL
LIN {X 0,Y 572.997,Z 745.78,A -85,B 0,C 180,E1 -2042.02,E2 -2042.02} C_VEL
LIN {X 0,Y 572.974,Z 749.058,A -85,B 0,C 180,E1 -2043.011,E2 -2043.011} C_VEL
LIN {X 0,Y 572.986,Z 751.22,A -85,B 0,C 180,E1 -2043.797,E2 -2043.797} C_VEL
LIN {X 0,Y 572.961,Z 754.374,A -85,B 0,C 180,E1 -2045.352,E2 -2045.352} C_VEL
LIN {X 0,Y 572.952,Z 756.102,A -85,B 0,C 180,E1 -2046.923,E2 -2046.923} C_VEL
LIN {X 0,Y 572.94,Z 756.426,A -85,B 0,C 180,E1 -2048.409,E2 -2048.409} C_VEL
LIN {X 0,Y 572.946,Z 755.462,A -85,B 0,C 180,E1 -2049.913,E2 -2049.913} C_VEL
LIN {X 0,Y 572.948,Z 753.212,A -85,B 0,C 180,E1 -2051.403,E2 -2051.403} C_VEL
LIN {X 0,Y 572.979,Z 749.655,A -85,B 0,C 180,E1 -2052.88,E2 -2052.88} C_VEL
LIN {X 0,Y 573.001,Z 744.753,A -85,B 0,C 180,E1 -2054.346,E2 -2054.346} C_VEL
LIN {X 0,Y 573.071,Z 738.401,A -85,B 0,C 180,E1 -2055.802,E2 -2055.802} C_VEL
LIN {X 0,Y 573.152,Z 730.451,A -85,B 0,C 180,E1 -2057.249,E2 -2057.249} C_VEL
LIN {X 0,Y 573.266,Z 722.022,A -85,B 0,C 180,E1 -2058.509,E2 -2058.509} C_VEL
LIN {X 0,Y 573.363,Z 711.946,A -85,B 0,C 180,E1 -2059.763,E2 -2059.763} C_VEL
LIN {X 0,Y 573.529,Z 701.712,A -85,B 0,C 180,E1 -2060.834,E2 -2060.834} C_VEL
LIN {X 0,Y 573.733,Z 689.538,A -85,B 0,C 180,E1 -2061.902,E2 -2061.902} C_VEL
LIN {X 0,Y 573.94,Z 676.559,A -85,B 0,C 180,E1 -2062.849,E2 -2062.849} C_VEL
LIN {X 0,Y 574.117,Z 664.307,A -85,B 0,C 180,E1 -2063.59,E2 -2063.59} C_VEL
LIN {X 0,Y 574.329,Z 649.962,A -85,B 0,C 180,E1 -2064.294,E2 -2064.294} C_VEL
LIN {X 0,Y 574.518,Z 634.892,A -85,B 0,C 180,E1 -2064.868,E2 -2064.868} C_VEL
LIN {X 0,Y 574.659,Z 619.825,A -85,B 0,C 180,E1 -2065.287,E2 -2065.287} C_VEL
LIN {X 0,Y 574.754,Z 605.403,A -85,B 0,C 180,E1 -2065.552,E2 -2065.552} C_VEL
LIN {X 0,Y 575.167,Z 453.234,A -85,B 0,C 180,E1 -2067.506,E2 -2067.506} C_VEL
LIN {X 0,Y 573.831,Z 445.901,A -85,B 0,C 180,E1 -2067.653,E2 -2067.653} C_VEL
LIN {X 0,Y 574.133,Z 425.183,A -85,B 0,C 180,E1 -2070.526,E2 -2070.526} C_VEL
LIN {X 0,Y 573.261,Z 419.706,A -85,B 0,C 180,E1 -2071.361,E2 -2071.361} C_VEL
LIN {X 0,Y 573.243,Z 419.708,A -85,B 0,C 180,E1 -2073.515,E2 -2073.515} C_VEL
LIN {X 0,Y 573.293,Z 419.701,A -85,B 0,C 180,E1 -2075.628,E2 -2075.628} C_VEL
LIN {X 0,Y 573.288,Z 419.694,A -85,B 0,C 180,E1 -2078.46,E2 -2078.46} C_VEL
LIN {X 0,Y 573.277,Z 419.698,A -85,B 0,C 180,E1 -2081.312,E2 -2081.312} C_VEL
LIN {X 0,Y 573.287,Z 419.694,A -85,B 0,C 180,E1 -2084.425,E2 -2084.425} C_VEL
LIN {X 0,Y 573.263,Z 419.699,A -85,B 0,C 180,E1 -2087.112,E2 -2087.112} C_VEL
LIN {X 0,Y 573.256,Z 419.7,A -85,B 0,C 180,E1 -2090.077,E2 -2090.077} C_VEL
LIN {X 0,Y 573.239,Z 419.702,A -85,B 0,C 180,E1 -2093.099,E2 -2093.099} C_VEL
LIN {X 0,Y 573.26,Z 419.702,A -85,B 0,C 180,E1 -2095.41,E2 -2095.41} C_VEL
LIN {X 0,Y 573.256,Z 419.7,A -85,B 0,C 180,E1 -2098.029,E2 -2098.029} C_VEL
LIN {X 0,Y 573.242,Z 419.699,A -85,B 0,C 180,E1 -2100.884,E2 -2100.884} C_VEL
LIN {X 0,Y 573.266,Z 419.702,A -85,B 0,C 180,E1 -2103.524,E2 -2103.524} C_VEL
LIN {X 0,Y 573.26,Z 419.7,A -85,B 0,C 180,E1 -2106.048,E2 -2106.048} C_VEL
LIN {X 0,Y 573.251,Z 419.696,A -85,B 0,C 180,E1 -2108.701,E2 -2108.701} C_VEL
LIN {X 0,Y 573.257,Z 419.706,A -85,B 0,C 180,E1 -2111.595,E2 -2111.595} C_VEL
LIN {X 0,Y 573.242,Z 419.699,A -85,B 0,C 180,E1 -2114.333,E2 -2114.333} C_VEL
LIN {X 0,Y 573.242,Z 419.704,A -85,B 0,C 180,E1 -2117.358,E2 -2117.358} C_VEL
LIN {X 0,Y 573.25,Z 419.698,A -85,B 0,C 180,E1 -2120.393,E2 -2120.393} C_VEL
LIN {X 0,Y 573.257,Z 419.698,A -85,B 0,C 180,E1 -2123.078,E2 -2123.078} C_VEL
LIN {X 0,Y 573.275,Z 419.704,A -85,B 0,C 180,E1 -2125.672,E2 -2125.672} C_VEL
LIN {X 0,Y 573.243,Z 419.7,A -85,B 0,C 180,E1 -2128.184,E2 -2128.184} C_VEL
LIN {X 0,Y 573.267,Z 419.694,A -85,B 0,C 180,E1 -2130.634,E2 -2130.634} C_VEL
LIN {X 0,Y 573.271,Z 419.702,A -85,B 0,C 180,E1 -2133.5,E2 -2133.5} C_VEL
LIN {X 0,Y 573.233,Z 419.7,A -85,B 0,C 180,E1 -2136.134,E2 -2136.134} C_VEL
LIN {X 0,Y 573.252,Z 419.699,A -85,B 0,C 180,E1 -2139.173,E2 -2139.173} C_VEL
LIN {X 0,Y 573.231,Z 419.706,A -85,B 0,C 180,E1 -2141.411,E2 -2141.411} C_VEL
LIN {X 0,Y 573.259,Z 419.704,A -85,B 0,C 180,E1 -2143.622,E2 -2143.622} C_VEL
LIN {X 0,Y 573.273,Z 419.703,A -85,B 0,C 180,E1 -2145.807,E2 -2145.807} C_VEL
LIN {X 0,Y 573.262,Z 419.695,A -85,B 0,C 180,E1 -2148.745,E2 -2148.745} C_VEL
LIN {X 0,Y 573.29,Z 419.698,A -85,B 0,C 180,E1 -2151.54,E2 -2151.54} C_VEL
LIN {X 0,Y 573.289,Z 419.693,A -85,B 0,C 180,E1 -2154.372,E2 -2154.372} C_VEL
LIN {X 0,Y 573.308,Z 419.696,A -85,B 0,C 180,E1 -2157.892,E2 -2157.892} C_VEL
LIN {X 0,Y 573.333,Z 419.687,A -85,B 0,C 180,E1 -2160.702,E2 -2160.702} C_VEL
LIN {X 0,Y 573.236,Z 419.706,A -85,B 0,C 180,E1 -2163.514,E2 -2163.514} C_VEL
LIN {X 0,Y 573.288,Z 419.699,A -85,B 0,C 180,E1 -2165.628,E2 -2165.628} C_VEL
LIN {X 0,Y 573.29,Z 419.693,A -85,B 0,C 180,E1 -2168.459,E2 -2168.459} C_VEL
LIN {X 0,Y 573.271,Z 419.698,A -85,B 0,C 180,E1 -2171.312,E2 -2171.312} C_VEL
LIN {X 0,Y 573.272,Z 419.698,A -85,B 0,C 180,E1 -2174.193,E2 -2174.193} C_VEL
LIN {X 0,Y 573.257,Z 419.698,A -85,B 0,C 180,E1 -2177.111,E2 -2177.111} C_VEL
LIN {X 0,Y 573.251,Z 419.701,A -85,B 0,C 180,E1 -2180.076,E2 -2180.076} C_VEL
LIN {X 0,Y 573.233,Z 419.701,A -85,B 0,C 180,E1 -2183.099,E2 -2183.099} C_VEL
LIN {X 0,Y 573.255,Z 419.702,A -85,B 0,C 180,E1 -2185.41,E2 -2185.41} C_VEL
LIN {X 0,Y 573.263,Z 419.701,A -85,B 0,C 180,E1 -2188.031,E2 -2188.031} C_VEL
LIN {X 0,Y 573.227,Z 419.7,A -85,B 0,C 180,E1 -2190.882,E2 -2190.882} C_VEL
LIN {X 0,Y 573.261,Z 419.703,A -85,B 0,C 180,E1 -2193.524,E2 -2193.524} C_VEL
LIN {X 0,Y 573.261,Z 419.701,A -85,B 0,C 180,E1 -2196.048,E2 -2196.048} C_VEL
LIN {X 0,Y 573.247,Z 419.698,A -85,B 0,C 180,E1 -2198.701,E2 -2198.701} C_VEL
LIN {X 0,Y 573.229,Z 419.706,A -85,B 0,C 180,E1 -2201.457,E2 -2201.457} C_VEL
LIN {X 0,Y 573.235,Z 419.701,A -85,B 0,C 180,E1 -2204.333,E2 -2204.333} C_VEL
LIN {X 0,Y 573.244,Z 419.703,A -85,B 0,C 180,E1 -2207.358,E2 -2207.358} C_VEL
LIN {X 0,Y 573.241,Z 419.7,A -85,B 0,C 180,E1 -2210.393,E2 -2210.393} C_VEL
LIN {X 0,Y 573.253,Z 419.699,A -85,B 0,C 180,E1 -2213.078,E2 -2213.078} C_VEL
LIN {X 0,Y 573.267,Z 419.705,A -85,B 0,C 180,E1 -2215.671,E2 -2215.671} C_VEL
LIN {X 0,Y 573.246,Z 419.703,A -85,B 0,C 180,E1 -2218.185,E2 -2218.185} C_VEL
LIN {X 0,Y 573.264,Z 419.699,A -85,B 0,C 180,E1 -2220.634,E2 -2220.634} C_VEL
LIN {X 0,Y 573.252,Z 419.703,A -85,B 0,C 180,E1 -2223.024,E2 -2223.024} C_VEL
LIN {X 0,Y 573.272,Z 419.775,A -85,B 0,C 180,E1 -2223.619,E2 -2223.619} C_VEL
LIN {X 0,Y 574.637,Z 425.981,A -85,B 0,C 180,E1 -2224.461,E2 -2224.461} C_VEL
LIN {X 0,Y 574.354,Z 447.83,A -85,B 0,C 180,E1 -2227.138,E2 -2227.138} C_VEL
LIN {X 0,Y 574.051,Z 472.575,A -85,B 0,C 180,E1 -2230.112,E2 -2230.112} C_VEL
LIN {X 0,Y 574.053,Z 475.248,A -85,B 0,C 180,E1 -2230.396,E2 -2230.396} C_VEL
LIN {X 0,Y 575.176,Z 481.409,A -85,B 0,C 180,E1 -2230.516,E2 -2230.516} C_VEL
LIN {X 0,Y 574.765,Z 640.973,A -85,B 0,C 180,E1 -2232.579,E2 -2232.579} C_VEL
LIN {X 0,Y 574.627,Z 656.699,A -85,B 0,C 180,E1 -2232.93,E2 -2232.93} C_VEL
LIN {X 0,Y 574.44,Z 672.037,A -85,B 0,C 180,E1 -2233.428,E2 -2233.428} C_VEL
LIN {X 0,Y 574.291,Z 685.764,A -85,B 0,C 180,E1 -2234.017,E2 -2234.017} C_VEL
LIN {X 0,Y 574.048,Z 699.238,A -85,B 0,C 180,E1 -2234.738,E2 -2234.738} C_VEL
LIN {X 0,Y 573.861,Z 712.813,A -85,B 0,C 180,E1 -2235.631,E2 -2235.631} C_VEL
LIN {X 0,Y 573.635,Z 725.346,A -85,B 0,C 180,E1 -2236.629,E2 -2236.629} C_VEL
LIN {X 0,Y 573.478,Z 735.746,A -85,B 0,C 180,E1 -2237.616,E2 -2237.616} C_VEL
LIN {X 0,Y 573.286,Z 745.768,A -85,B 0,C 180,E1 -2238.734,E2 -2238.734} C_VEL
LIN {X 0,Y 573.243,Z 754.855,A -85,B 0,C 180,E1 -2239.938,E2 -2239.938} C_VEL
LIN {X 0,Y 573.133,Z 762.731,A -85,B 0,C 180,E1 -2241.183,E2 -2241.183} C_VEL
LIN {X 0,Y 573.075,Z 770.088,A -85,B 0,C 180,E1 -2242.601,E2 -2242.601} C_VEL
LIN {X 0,Y 573.04,Z 775.922,A -85,B 0,C 180,E1 -2244.016,E2 -2244.016} C_VEL
LIN {X 0,Y 572.951,Z 779.384,A -85,B 0,C 180,E1 -2245.074,E2 -2245.074} C_VEL
LIN {X 0,Y 573.004,Z 782.888,A -85,B 0,C 180,E1 -2246.484,E2 -2246.484} C_VEL
LIN {X 0,Y 572.935,Z 785.192,A -85,B 0,C 180,E1 -2247.891,E2 -2247.891} C_VEL
LIN {X 0,Y 572.938,Z 786.349,A -85,B 0,C 180,E1 -2249.297,E2 -2249.297} C_VEL
LIN {X 0,Y 572.938,Z 786.349,A -85,B 0,C 180,E1 -2250.702,E2 -2250.702} C_VEL
LIN {X 0,Y 572.935,Z 785.192,A -85,B 0,C 180,E1 -2252.109,E2 -2252.109} C_VEL
LIN {X 0,Y 573.004,Z 782.888,A -85,B 0,C 180,E1 -2253.515,E2 -2253.515} C_VEL
LIN {X 0,Y 572.951,Z 779.386,A -85,B 0,C 180,E1 -2254.925,E2 -2254.925} C_VEL
LIN {X 0,Y 573.012,Z 774.61,A -85,B 0,C 180,E1 -2256.337,E2 -2256.337} C_VEL
LIN {X 0,Y 573.095,Z 768.426,A -85,B 0,C 180,E1 -2257.752,E2 -2257.752} C_VEL
LIN {X 0,Y 573.136,Z 760.652,A -85,B 0,C 180,E1 -2259.172,E2 -2259.172} C_VEL
LIN {X 0,Y 573.27,Z 752.373,A -85,B 0,C 180,E1 -2260.417,E2 -2260.417} C_VEL
LIN {X 0,Y 573.385,Z 742.396,A -85,B 0,C 180,E1 -2261.668,E2 -2261.668} C_VEL
LIN {X 0,Y 573.567,Z 732.195,A -85,B 0,C 180,E1 -2262.741,E2 -2262.741} C_VEL
LIN {X 0,Y 573.742,Z 720.026,A -85,B 0,C 180,E1 -2263.819,E2 -2263.819} C_VEL
LIN {X 0,Y 573.959,Z 706.911,A -85,B 0,C 180,E1 -2264.781,E2 -2264.781} C_VEL
LIN {X 0,Y 574.109,Z 694.527,A -85,B 0,C 180,E1 -2265.532,E2 -2265.532} C_VEL
LIN {X 0,Y 574.352,Z 679.846,A -85,B 0,C 180,E1 -2266.254,E2 -2266.254} C_VEL
LIN {X 0,Y 574.515,Z 666.932,A -85,B 0,C 180,E1 -2266.752,E2 -2266.752} C_VEL
